LIN {X 0,Y 516.913,Z 376.098,A -85,B 0,C 180,E1 -4916.12,E2 -4916.12} C_VEL
LIN {X 0,Y 516.895,Z 376.101,A -85,B 0,C 180,E1 -4918.935,E2 -4918.935} C_VEL
LIN {X 0,Y 516.92,Z 376.096,A -85,B 0,C 180,E1 -4921.584,E2 -4921.584} C_VEL
LIN {X 0,Y 516.937,Z 376.095,A -85,B 0,C 180,E1 -4924.21,E2 -4924.21} C_VEL
LIN {X 0,Y 516.871,Z 376.104,A -85,B 0,C 180,E1 -4926.775,E2 -4926.775} C_VEL
LIN {X 0,Y 516.945,Z 376.094,A -85,B 0,C 180,E1 -4929.731,E2 -4929.731} C_VEL
LIN {X 0,Y 516.925,Z 376.098,A -85,B 0,C 180,E1 -4932.595,E2 -4932.595} C_VEL
LIN {X 0,Y 516.947,Z 376.094,A -85,B 0,C 180,E1 -4935.029,E2 -4935.029} C_VEL
LIN {X 0,Y 516.884,Z 376.104,A -85,B 0,C 180,E1 -4938.231,E2 -4938.231} C_VEL
LIN {X 0,Y 516.594,Z 376.439,A -85,B 0,C 180,E1 -4940.603,E2 -4940.603} C_VEL
LIN {X 0,Y 516.577,Z 379.88,A -85,B 0,C 180,E1 -4943.75,E2 -4943.75} C_VEL
LIN {X 0,Y 516.567,Z 382.466,A -85,B 0,C 180,E1 -4946.098,E2 -4946.098} C_VEL
LIN {X 0,Y 516.432,Z 386.765,A -85,B 0,C 180,E1 -4949.999,E2 -4949.999} C_VEL
LIN {X 0,Y 516.446,Z 391.091,A -85,B 0,C 180,E1 -4953.9,E2 -4953.9} C_VEL
LIN {X 0,Y 516.401,Z 394.057,A -85,B 0,C 180,E1 -4956.536,E2 -4956.536} C_VEL
LIN {X 0,Y 516.278,Z 397.014,A -85,B 0,C 180,E1 -4959.202,E2 -4959.202} C_VEL
LIN {X 0,Y 518.475,Z 408.871,A -85,B 0,C 180,E1 -4959.581,E2 -4959.581} C_VEL
LIN {X 0,Y 518.24,Z 422.351,A -85,B 0,C 180,E1 -4960.103,E2 -4960.103} C_VEL
LIN {X 0,Y 517.891,Z 434.499,A -85,B 0,C 180,E1 -4960.752,E2 -4960.752} C_VEL
LIN {X 0,Y 517.599,Z 446.016,A -85,B 0,C 180,E1 -4961.551,E2 -4961.551} C_VEL
LIN {X 0,Y 517.28,Z 455.69,A -85,B 0,C 180,E1 -4962.386,E2 -4962.386} C_VEL
LIN {X 0,Y 517.014,Z 464.898,A -85,B 0,C 180,E1 -4963.359,E2 -4963.359} C_VEL
LIN {X 0,Y 516.749,Z 474.087,A -85,B 0,C 180,E1 -4964.571,E2 -4964.571} C_VEL
LIN {X 0,Y 516.599,Z 481.479,A -85,B 0,C 180,E1 -4965.787,E2 -4965.787} C_VEL
LIN {X 0,Y 516.454,Z 487.37,A -85,B 0,C 180,E1 -4967.01,E2 -4967.01} C_VEL
LIN {X 0,Y 516.35,Z 491.98,A -85,B 0,C 180,E1 -4968.241,E2 -4968.241} C_VEL
LIN {X 0,Y 516.29,Z 494.408,A -85,B 0,C 180,E1 -4969.067,E2 -4969.067} C_VEL
LIN {X 0,Y 516.231,Z 496.687,A -85,B 0,C 180,E1 -4970.054,E2 -4970.054} C_VEL
LIN {X 0,Y 516.201,Z 498.869,A -85,B 0,C 180,E1 -4971.566,E2 -4971.566} C_VEL
LIN {X 0,Y 516.214,Z 499.464,A -85,B 0,C 180,E1 -4972.406,E2 -4972.406} C_VEL
LIN {X 0,Y 516.183,Z 499.561,A -85,B 0,C 180,E1 -4973.254,E2 -4973.254} C_VEL
LIN {X 0,Y 516.199,Z 499.165,A -85,B 0,C 180,E1 -4974.189,E2 -4974.189} C_VEL
LIN {X 0,Y 516.2,Z 498.417,A -85,B 0,C 180,E1 -4974.963,E2 -4974.963} C_VEL
LIN {X 0,Y 516.222,Z 496.702,A -85,B 0,C 180,E1 -4976.033,E2 -4976.033} C_VEL
LIN {X 0,Y 516.305,Z 494.141,A -85,B 0,C 180,E1 -4977.127,E2 -4977.127} C_VEL
LIN {X 0,Y 516.383,Z 489.92,A -85,B 0,C 180,E1 -4978.445,E2 -4978.445} C_VEL
LIN {X 0,Y 516.516,Z 484.125,A -85,B 0,C 180,E1 -4979.794,E2 -4979.794} C_VEL
LIN {X 0,Y 516.715,Z 476.736,A -85,B 0,C 180,E1 -4981.119,E2 -4981.119} C_VEL
LIN {X 0,Y 516.92,Z 469.222,A -85,B 0,C 180,E1 -4982.2,E2 -4982.2} C_VEL
LIN {X 0,Y 517.194,Z 460.061,A -85,B 0,C 180,E1 -4983.271,E2 -4983.271} C_VEL
LIN {X 0,Y 517.481,Z 449.897,A -85,B 0,C 180,E1 -4984.228,E2 -4984.228} C_VEL
LIN {X 0,Y 517.778,Z 439.926,A -85,B 0,C 180,E1 -4984.989,E2 -4984.989} C_VEL
LIN {X 0,Y 518.075,Z 428.588,A -85,B 0,C 180,E1 -4985.682,E2 -4985.682} C_VEL
LIN {X 0,Y 518.328,Z 415.979,A -85,B 0,C 180,E1 -4986.262,E2 -4986.262} C_VEL
LIN {X 0,Y 518.286,Z 407.164,A -85,B 0,C 180,E1 -4986.574,E2 -4986.574} C_VEL
LIN {X 0,Y 516.296,Z 397.126,A -85,B 0,C 180,E1 -4986.895,E2 -4986.895} C_VEL
LIN {X 0,Y 516.309,Z 393.355,A -85,B 0,C 180,E1 -4990.335,E2 -4990.335} C_VEL
LIN {X 0,Y 516.37,Z 390.564,A -85,B 0,C 180,E1 -4992.881,E2 -4992.881} C_VEL
LIN {X 0,Y 516.411,Z 388.218,A -85,B 0,C 180,E1 -4995.044,E2 -4995.044} C_VEL
LIN {X 0,Y 516.446,Z 384.839,A -85,B 0,C 180,E1 -4998.179,E2 -4998.179} C_VEL
LIN {X 0,Y 516.457,Z 381.512,A -85,B 0,C 180,E1 -5001.246,E2 -5001.246} C_VEL
LIN {X 0,Y 516.553,Z 378.293,A -85,B 0,C 180,E1 -5004.194,E2 -5004.194} C_VEL
LIN {X 0,Y 516.601,Z 376.21,A -85,B 0,C 180,E1 -5006.098,E2 -5006.098} C_VEL
LIN {X 0,Y 516.861,Z 376.104,A -85,B 0,C 180,E1 -5008.937,E2 -5008.937} C_VEL
LIN {X 0,Y 516.907,Z 376.097,A -85,B 0,C 180,E1 -5011.584,E2 -5011.584} C_VEL
LIN {X 0,Y 516.915,Z 376.097,A -85,B 0,C 180,E1 -5014.21,E2 -5014.21} C_VEL
LIN {X 0,Y 516.885,Z 376.101,A -85,B 0,C 180,E1 -5016.777,E2 -5016.777} C_VEL
LIN {X 0,Y 516.92,Z 376.095,A -85,B 0,C 180,E1 -5019.73,E2 -5019.73} C_VEL
LIN {X 0,Y 516.911,Z 376.096,A -85,B 0,C 180,E1 -5022.596,E2 -5022.596} C_VEL
LIN {X 0,Y 516.921,Z 376.095,A -85,B 0,C 180,E1 -5025.03,E2 -5025.03} C_VEL
LIN {X 0,Y 516.983,Z 376.088,A -85,B 0,C 180,E1 -5028.234,E2 -5028.234} C_VEL
LIN {X 0,Y 516.953,Z 376.094,A -85,B 0,C 180,E1 -5031.399,E2 -5031.399} C_VEL
LIN {X 0,Y 517.047,Z 376.08,A -85,B 0,C 180,E1 -5034.54,E2 -5034.54} C_VEL
LIN {X 0,Y 517.07,Z 376.077,A -85,B 0,C 180,E1 -5037.663,E2 -5037.663} C_VEL
LIN {X 0,Y 517.077,Z 376.079,A -85,B 0,C 180,E1 -5040.779,E2 -5040.779} C_VEL
LIN {X 0,Y 517.026,Z 376.083,A -85,B 0,C 180,E1 -5043.117,E2 -5043.117} C_VEL
LIN {X 0,Y 516.991,Z 376.09,A -85,B 0,C 180,E1 -5046.243,E2 -5046.243} C_VEL
LIN {X 0,Y 516.937,Z 376.093,A -85,B 0,C 180,E1 -5049.39,E2 -5049.39} C_VEL
LIN {X 0,Y 516.962,Z 376.092,A -85,B 0,C 180,E1 -5051.825,E2 -5051.825} C_VEL
LIN {X 0,Y 516.923,Z 376.095,A -85,B 0,C 180,E1 -5055.147,E2 -5055.147} C_VEL
LIN {X 0,Y 516.907,Z 376.1,A -85,B 0,C 180,E1 -5058.223,E2 -5058.223} C_VEL
LIN {X 0,Y 516.898,Z 376.099,A -85,B 0,C 180,E1 -5060.702,E2 -5060.702} C_VEL
LIN {X 0,Y 516.888,Z 376.1,A -85,B 0,C 180,E1 -5063.223,E2 -5063.223} C_VEL
LIN {X 0,Y 516.926,Z 376.098,A -85,B 0,C 180,E1 -5066.198,E2 -5066.198} C_VEL
LIN {X 0,Y 516.905,Z 376.101,A -85,B 0,C 180,E1 -5069.306,E2 -5069.306} C_VEL
LIN {X 0,Y 516.884,Z 376.1,A -85,B 0,C 180,E1 -5072.546,E2 -5072.546} C_VEL
LIN {X 0,Y 516.868,Z 376.102,A -85,B 0,C 180,E1 -5075.334,E2 -5075.334} C_VEL
LIN {X 0,Y 516.869,Z 376.102,A -85,B 0,C 180,E1 -5077.945,E2 -5077.945} C_VEL
LIN {X 0,Y 516.894,Z 376.101,A -85,B 0,C 180,E1 -5080.741,E2 -5080.741} C_VEL
LIN {X 0,Y 516.869,Z 376.108,A -85,B 0,C 180,E1 -5083.905,E2 -5083.905} C_VEL
LIN {X 0,Y 516.87,Z 376.106,A -85,B 0,C 180,E1 -5086.109,E2 -5086.109} C_VEL
LIN {X 0,Y 516.894,Z 376.103,A -85,B 0,C 180,E1 -5089.262,E2 -5089.262} C_VEL
LIN {X 0,Y 516.908,Z 376.193,A -85,B 0,C 180,E1 -5091.229,E2 -5091.229} C_VEL
LIN {X 0,Y 518.065,Z 382.766,A -85,B 0,C 180,E1 -5093.838,E2 -5093.838} C_VEL
LIN {X 0,Y 518.075,Z 388.22,A -85,B 0,C 180,E1 -5095.843,E2 -5095.843} C_VEL
LIN {X 0,Y 517.76,Z 397.502,A -85,B 0,C 180,E1 -5098.951,E2 -5098.951} C_VEL
LIN {X 0,Y 517.58,Z 406.694,A -85,B 0,C 180,E1 -5101.959,E2 -5101.959} C_VEL
LIN {X 0,Y 517.315,Z 414.964,A -85,B 0,C 180,E1 -5104.665,E2 -5104.665} C_VEL
LIN {X 0,Y 517.11,Z 424.231,A -85,B 0,C 180,E1 -5107.635,E2 -5107.635} C_VEL
LIN {X 0,Y 516.902,Z 433.498,A -85,B 0,C 180,E1 -5110.544,E2 -5110.544} C_VEL
LIN {X 0,Y 516.709,Z 442.766,A -85,B 0,C 180,E1 -5113.405,E2 -5113.405} C_VEL
LIN {X 0,Y 516.577,Z 451.536,A -85,B 0,C 180,E1 -5116.078,E2 -5116.078} C_VEL
LIN {X 0,Y 518.522,Z 464.249,A -85,B 0,C 180,E1 -5116.431,E2 -5116.431} C_VEL
LIN {X 0,Y 518.314,Z 475.818,A -85,B 0,C 180,E1 -5116.824,E2 -5116.824} C_VEL
LIN {X 0,Y 517.995,Z 487.442,A -85,B 0,C 180,E1 -5117.364,E2 -5117.364} C_VEL
LIN {X 0,Y 517.684,Z 499.584,A -85,B 0,C 180,E1 -5118.11,E2 -5118.11} C_VEL
LIN {X 0,Y 517.42,Z 510.283,A -85,B 0,C 180,E1 -5118.941,E2 -5118.941} C_VEL
LIN {X 0,Y 517.081,Z 519.555,A -85,B 0,C 180,E1 -5119.825,E2 -5119.825} C_VEL
LIN {X 0,Y 516.866,Z 528.004,A -85,B 0,C 180,E1 -5120.808,E2 -5120.808} C_VEL
LIN {X 0,Y 516.639,Z 536.247,A -85,B 0,C 180,E1 -5121.987,E2 -5121.987} C_VEL
LIN {X 0,Y 516.478,Z 543.085,A -85,B 0,C 180,E1 -5123.203,E2 -5123.203} C_VEL
LIN {X 0,Y 516.405,Z 548.956,A -85,B 0,C 180,E1 -5124.535,E2 -5124.535} C_VEL
LIN {X 0,Y 516.343,Z 552.899,A -85,B 0,C 180,E1 -5125.708,E2 -5125.708} C_VEL
LIN {X 0,Y 516.282,Z 555.811,A -85,B 0,C 180,E1 -5126.88,E2 -5126.88} C_VEL
LIN {X 0,Y 516.261,Z 557.199,A -85,B 0,C 180,E1 -5127.661,E2 -5127.661} C_VEL
LIN {X 0,Y 516.16,Z 558.786,A -85,B 0,C 180,E1 -5129.221,E2 -5129.221} C_VEL
LIN {X 0,Y 516.154,Z 559,A -85,B 0,C 180,E1 -5130.001,E2 -5130.001} C_VEL
LIN {X 0,Y 516.192,Z 558.184,A -85,B 0,C 180,E1 -5131.562,E2 -5131.562} C_VEL
LIN {X 0,Y 516.262,Z 557.196,A -85,B 0,C 180,E1 -5132.342,E2 -5132.342} C_VEL
LIN {X 0,Y 516.283,Z 555.807,A -85,B 0,C 180,E1 -5133.123,E2 -5133.123} C_VEL
LIN {X 0,Y 516.344,Z 552.892,A -85,B 0,C 180,E1 -5134.295,E2 -5134.295} C_VEL
LIN {X 0,Y 516.406,Z 548.944,A -85,B 0,C 180,E1 -5135.468,E2 -5135.468} C_VEL
LIN {X 0,Y 516.488,Z 543.025,A -85,B 0,C 180,E1 -5136.809,E2 -5136.809} C_VEL
LIN {X 0,Y 516.642,Z 536.228,A -85,B 0,C 180,E1 -5138.016,E2 -5138.016} C_VEL
LIN {X 0,Y 516.871,Z 527.981,A -85,B 0,C 180,E1 -5139.195,E2 -5139.195} C_VEL
LIN {X 0,Y 517.08,Z 519.526,A -85,B 0,C 180,E1 -5140.178,E2 -5140.178} C_VEL
LIN {X 0,Y 517.434,Z 509.081,A -85,B 0,C 180,E1 -5141.161,E2 -5141.161} C_VEL
LIN {X 0,Y 517.7,Z 497.781,A -85,B 0,C 180,E1 -5142.016,E2 -5142.016} C_VEL
LIN {X 0,Y 517.992,Z 487.386,A -85,B 0,C 180,E1 -5142.639,E2 -5142.639} C_VEL
LIN {X 0,Y 518.284,Z 475.731,A -85,B 0,C 180,E1 -5143.179,E2 -5143.179} C_VEL
LIN {X 0,Y 518.421,Z 462.758,A -85,B 0,C 180,E1 -5143.613,E2 -5143.613} C_VEL
LIN {X 0,Y 516.577,Z 451.526,A -85,B 0,C 180,E1 -5143.925,E2 -5143.925} C_VEL
LIN {X 0,Y 516.715,Z 442.755,A -85,B 0,C 180,E1 -5146.598,E2 -5146.598} C_VEL
LIN {X 0,Y 516.91,Z 433.488,A -85,B 0,C 180,E1 -5149.459,E2 -5149.459} C_VEL
LIN {X 0,Y 517.102,Z 423.961,A -85,B 0,C 180,E1 -5152.452,E2 -5152.452} C_VEL
LIN {X 0,Y 517.376,Z 413.63,A -85,B 0,C 180,E1 -5155.766,E2 -5155.766} C_VEL
LIN {X 0,Y 517.604,Z 404.3,A -85,B 0,C 180,E1 -5158.818,E2 -5158.818} C_VEL
LIN {X 0,Y 517.882,Z 394.893,A -85,B 0,C 180,E1 -5161.956,E2 -5161.956} C_VEL
LIN {X 0,Y 518.147,Z 386.815,A -85,B 0,C 180,E1 -5164.729,E2 -5164.729} C_VEL
LIN {X 0,Y 518.059,Z 382.767,A -85,B 0,C 180,E1 -5166.167,E2 -5166.167} C_VEL
LIN {X 0,Y 516.886,Z 376.104,A -85,B 0,C 180,E1 -5168.836,E2 -5168.836} C_VEL
LIN {X 0,Y 516.917,Z 376.097,A -85,B 0,C 180,E1 -5171.776,E2 -5171.776} C_VEL
LIN {X 0,Y 516.901,Z 376.1,A -85,B 0,C 180,E1 -5175.007,E2 -5175.007} C_VEL
LIN {X 0,Y 516.919,Z 376.098,A -85,B 0,C 180,E1 -5178.399,E2 -5178.399} C_VEL
LIN {X 0,Y 516.885,Z 376.102,A -85,B 0,C 180,E1 -5181.284,E2 -5181.284} C_VEL
LIN {X 0,Y 516.876,Z 376.103,A -85,B 0,C 180,E1 -5184.22,E2 -5184.22} C_VEL
LIN {X 0,Y 516.886,Z 376.102,A -85,B 0,C 180,E1 -5187.052,E2 -5187.052} C_VEL
LIN {X 0,Y 516.897,Z 376.099,A -85,B 0,C 180,E1 -5189.796,E2 -5189.796} C_VEL
LIN {X 0,Y 516.93,Z 376.096,A -85,B 0,C 180,E1 -5192.467,E2 -5192.467} C_VEL
LIN {X 0,Y 516.913,Z 376.099,A -85,B 0,C 180,E1 -5195.072,E2 -5195.072} C_VEL
LIN {X 0,Y 516.89,Z 376.102,A -85,B 0,C 180,E1 -5198.462,E2 -5198.462} C_VEL
LIN {X 0,Y 516.907,Z 376.099,A -85,B 0,C 180,E1 -5200.955,E2 -5200.955} C_VEL
LIN {X 0,Y 516.918,Z 376.097,A -85,B 0,C 180,E1 -5203.41,E2 -5203.41} C_VEL
LIN {X 0,Y 516.899,Z 376.1,A -85,B 0,C 180,E1 -5205.834,E2 -5205.834} C_VEL
LIN {X 0,Y 516.97,Z 376.091,A -85,B 0,C 180,E1 -5208.234,E2 -5208.234} C_VEL
LIN {X 0,Y 516.974,Z 376.089,A -85,B 0,C 180,E1 -5211.4,E2 -5211.4} C_VEL
LIN {X 0,Y 517.013,Z 376.086,A -85,B 0,C 180,E1 -5213.757,E2 -5213.757} C_VEL
LIN {X 0,Y 517.087,Z 376.076,A -85,B 0,C 180,E1 -5217.663,E2 -5217.663} C_VEL
LIN {X 0,Y 517.095,Z 376.075,A -85,B 0,C 180,E1 -5220.779,E2 -5220.779} C_VEL
LIN {X 0,Y 517.016,Z 376.085,A -85,B 0,C 180,E1 -5223.117,E2 -5223.117} C_VEL
LIN {X 0,Y 517.007,Z 376.088,A -85,B 0,C 180,E1 -5226.243,E2 -5226.243} C_VEL
LIN {X 0,Y 516.957,Z 376.093,A -85,B 0,C 180,E1 -5229.389,E2 -5229.389} C_VEL
LIN {X 0,Y 516.956,Z 376.093,A -85,B 0,C 180,E1 -5231.807,E2 -5231.807} C_VEL
LIN {X 0,Y 516.949,Z 376.093,A -85,B 0,C 180,E1 -5235.146,E2 -5235.146} C_VEL
LIN {X 0,Y 516.928,Z 376.096,A -85,B 0,C 180,E1 -5238.222,E2 -5238.222} C_VEL
LIN {X 0,Y 516.916,Z 376.098,A -85,B 0,C 180,E1 -5240.701,E2 -5240.701} C_VEL
LIN {X 0,Y 516.908,Z 376.099,A -85,B 0,C 180,E1 -5244.072,E2 -5244.072} C_VEL
LIN {X 0,Y 516.93,Z 376.094,A -85,B 0,C 180,E1 -5246.658,E2 -5246.658} C_VEL
LIN {X 0,Y 516.915,Z 376.098,A -85,B 0,C 180,E1 -5249.523,E2 -5249.523} C_VEL
LIN {X 0,Y 516.9,Z 376.099,A -85,B 0,C 180,E1 -5252.543,E2 -5252.543} C_VEL
LIN {X 0,Y 516.87,Z 376.106,A -85,B 0,C 180,E1 -5255.329,E2 -5255.329} C_VEL
LIN {X 0,Y 516.884,Z 376.101,A -85,B 0,C 180,E1 -5257.942,E2 -5257.942} C_VEL
LIN {X 0,Y 516.887,Z 376.102,A -85,B 0,C 180,E1 -5260.741,E2 -5260.741} C_VEL
LIN {X 0,Y 516.887,Z 376.102,A -85,B 0,C 180,E1 -5262.831,E2 -5262.831} C_VEL
LIN {X 0,Y 516.9,Z 376.1,A -85,B 0,C 180,E1 -5265.007,E2 -5265.007} C_VEL
LIN {X 0,Y 516.92,Z 376.096,A -85,B 0,C 180,E1 -5268.398,E2 -5268.398} C_VEL
LIN {X 0,Y 516.887,Z 376.1,A -85,B 0,C 180,E1 -5270.301,E2 -5270.301} C_VEL
LIN {X 0,Y 516.216,Z 376.187,A -85,B 0,C 180,E1 -5270.951,E2 -5270.951} C_VEL
LIN {X 0,Y 513.369,Z 376.542,A -85,B 0,C 180,E1 -5272.007,E2 -5272.007} C_VEL
LIN {X 0,Y 510.959,Z 376.843,A -85,B 0,C 180,E1 -5272.857,E2 -5272.857} C_VEL
LIN {X 0,Y 509.915,Z 376.971,A -85,B 0,C 180,E1 -5273.514,E2 -5273.514} C_VEL
LIN {X 0,Y 509.825,Z 376.981,A -85,B 0,C 180,E1 -5273.736,E2 -5273.736} C_VEL
LIN {X 0,Y 509.864,Z 376.976,A -85,B 0,C 180,E1 -5276.538,E2 -5276.538} C_VEL
LIN {X 0,Y 509.848,Z 376.978,A -85,B 0,C 180,E1 -5279.333,E2 -5279.333} C_VEL
LIN {X 0,Y 509.895,Z 376.971,A -85,B 0,C 180,E1 -5282.054,E2 -5282.054} C_VEL
LIN {X 0,Y 509.882,Z 376.974,A -85,B 0,C 180,E1 -5284.703,E2 -5284.703} C_VEL
LIN {X 0,Y 509.832,Z 376.98,A -85,B 0,C 180,E1 -5287.457,E2 -5287.457} C_VEL
LIN {X 0,Y 509.922,Z 376.968,A -85,B 0,C 180,E1 -5289.844,E2 -5289.844} C_VEL
LIN {X 0,Y 509.885,Z 376.973,A -85,B 0,C 180,E1 -5293.174,E2 -5293.174} C_VEL
LIN {X 0,Y 509.867,Z 376.975,A -85,B 0,C 180,E1 -5295.633,E2 -5295.633} C_VEL
LIN {X 0,Y 509.848,Z 376.98,A -85,B 0,C 180,E1 -5298.154,E2 -5298.154} C_VEL
LIN {X 0,Y 509.521,Z 377.021,A -85,B 0,C 180,E1 -5300.471,E2 -5300.471} C_VEL
LIN {X 0,Y 509.527,Z 380.47,A -85,B 0,C 180,E1 -5303.663,E2 -5303.663} C_VEL
LIN {X 0,Y 509.519,Z 383.053,A -85,B 0,C 180,E1 -5306.044,E2 -5306.044} C_VEL
LIN {X 0,Y 509.359,Z 387.412,A -85,B 0,C 180,E1 -5309.998,E2 -5309.998} C_VEL
LIN {X 0,Y 509.371,Z 391.778,A -85,B 0,C 180,E1 -5313.954,E2 -5313.954} C_VEL
LIN {X 0,Y 509.347,Z 394.758,A -85,B 0,C 180,E1 -5316.555,E2 -5316.555} C_VEL
LIN {X 0,Y 509.21,Z 397.44,A -85,B 0,C 180,E1 -5319.006,E2 -5319.006} C_VEL
LIN {X 0,Y 511.522,Z 409.074,A -85,B 0,C 180,E1 -5319.388,E2 -5319.388} C_VEL
LIN {X 0,Y 511.364,Z 421.956,A -85,B 0,C 180,E1 -5319.89,E2 -5319.89} C_VEL
LIN {X 0,Y 511.001,Z 433.55,A -85,B 0,C 180,E1 -5320.498,E2 -5320.498} C_VEL
LIN {X 0,Y 510.697,Z 445.317,A -85,B 0,C 180,E1 -5321.307,E2 -5321.307} C_VEL
LIN {X 0,Y 510.32,Z 455.958,A -85,B 0,C 180,E1 -5322.225,E2 -5322.225} C_VEL
LIN {X 0,Y 510.067,Z 464.568,A -85,B 0,C 180,E1 -5323.139,E2 -5323.139} C_VEL
LIN {X 0,Y 509.792,Z 472.538,A -85,B 0,C 180,E1 -5324.162,E2 -5324.162} C_VEL
LIN {X 0,Y 509.595,Z 480.277,A -85,B 0,C 180,E1 -5325.394,E2 -5325.394} C_VEL
LIN {X 0,Y 509.425,Z 485.575,A -85,B 0,C 180,E1 -5326.426,E2 -5326.426} C_VEL
LIN {X 0,Y 509.304,Z 491.125,A -85,B 0,C 180,E1 -5327.797,E2 -5327.797} C_VEL
LIN {X 0,Y 509.224,Z 494.601,A -85,B 0,C 180,E1 -5328.923,E2 -5328.923} C_VEL
LIN {X 0,Y 509.134,Z 497.43,A -85,B 0,C 180,E1 -5330.186,E2 -5330.186} C_VEL
LIN {X 0,Y 509.119,Z 498.746,A -85,B 0,C 180,E1 -5331.031,E2 -5331.031} C_VEL
LIN {X 0,Y 509.123,Z 499.873,A -85,B 0,C 180,E1 -5332.35,E2 -5332.35} C_VEL
LIN {X 0,Y 509.104,Z 499.927,A -85,B 0,C 180,E1 -5333.597,E2 -5333.597} C_VEL
LIN {X 0,Y 509.106,Z 499.39,A -85,B 0,C 180,E1 -5334.463,E2 -5334.463} C_VEL
LIN {X 0,Y 509.107,Z 498.37,A -85,B 0,C 180,E1 -5335.335,E2 -5335.335} C_VEL
LIN {X 0,Y 509.192,Z 495.915,A -85,B 0,C 180,E1 -5336.65,E2 -5336.65} C_VEL
LIN {X 0,Y 509.275,Z 492.238,A -85,B 0,C 180,E1 -5337.98,E2 -5337.98} C_VEL
LIN {X 0,Y 509.401,Z 487.436,A -85,B 0,C 180,E1 -5339.259,E2 -5339.259} C_VEL
LIN {X 0,Y 509.569,Z 480.412,A -85,B 0,C 180,E1 -5340.682,E2 -5340.682} C_VEL
LIN {X 0,Y 509.823,Z 473.326,A -85,B 0,C 180,E1 -5341.82,E2 -5341.82} C_VEL
LIN {X 0,Y 510.065,Z 465.228,A -85,B 0,C 180,E1 -5342.883,E2 -5342.883} C_VEL
LIN {X 0,Y 510.398,Z 455.733,A -85,B 0,C 180,E1 -5343.892,E2 -5343.892} C_VEL
LIN {X 0,Y 510.72,Z 444.893,A -85,B 0,C 180,E1 -5344.823,E2 -5344.823} C_VEL
LIN {X 0,Y 511.012,Z 434.442,A -85,B 0,C 180,E1 -5345.542,E2 -5345.542} C_VEL
LIN {X 0,Y 511.318,Z 423.016,A -85,B 0,C 180,E1 -5346.159,E2 -5346.159} C_VEL
LIN {X 0,Y 511.585,Z 410.272,A -85,B 0,C 180,E1 -5346.664,E2 -5346.664} C_VEL
LIN {X 0,Y 510.149,Z 401.591,A -85,B 0,C 180,E1 -5346.962,E2 -5346.962} C_VEL
LIN {X 0,Y 509.214,Z 397.595,A -85,B 0,C 180,E1 -5347.084,E2 -5347.084} C_VEL
LIN {X 0,Y 509.252,Z 393.912,A -85,B 0,C 180,E1 -5350.435,E2 -5350.435} C_VEL
LIN {X 0,Y 509.339,Z 390.438,A -85,B 0,C 180,E1 -5353.62,E2 -5353.62} C_VEL
LIN {X 0,Y 509.364,Z 387.478,A -85,B 0,C 180,E1 -5356.379,E2 -5356.379} C_VEL
LIN {X 0,Y 509.401,Z 384.264,A -85,B 0,C 180,E1 -5359.356,E2 -5359.356} C_VEL
LIN {X 0,Y 509.453,Z 380.728,A -85,B 0,C 180,E1 -5362.628,E2 -5362.628} C_VEL
LIN {X 0,Y 509.527,Z 377.543,A -85,B 0,C 180,E1 -5365.562,E2 -5365.562} C_VEL
LIN {X 0,Y 509.574,Z 377.015,A -85,B 0,C 180,E1 -5366.518,E2 -5366.518} C_VEL
LIN {X 0,Y 509.823,Z 376.982,A -85,B 0,C 180,E1 -5369.333,E2 -5369.333} C_VEL
LIN {X 0,Y 509.877,Z 376.974,A -85,B 0,C 180,E1 -5372.054,E2 -5372.054} C_VEL
LIN {X 0,Y 509.865,Z 376.976,A -85,B 0,C 180,E1 -5374.703,E2 -5374.703} C_VEL
LIN {X 0,Y 509.864,Z 376.976,A -85,B 0,C 180,E1 -5377.441,E2 -5377.441} C_VEL
LIN {X 0,Y 509.897,Z 376.969,A -85,B 0,C 180,E1 -5379.844,E2 -5379.844} C_VEL
LIN {X 0,Y 509.867,Z 376.978,A -85,B 0,C 180,E1 -5383.174,E2 -5383.174} C_VEL
LIN {X 0,Y 509.845,Z 376.978,A -85,B 0,C 180,E1 -5385.634,E2 -5385.634} C_VEL
LIN {X 0,Y 509.907,Z 376.97,A -85,B 0,C 180,E1 -5388.874,E2 -5388.874} C_VEL
LIN {X 0,Y 509.931,Z 376.966,A -85,B 0,C 180,E1 -5392.078,E2 -5392.078} C_VEL
LIN {X 0,Y 509.993,Z 376.959,A -85,B 0,C 180,E1 -5394.464,E2 -5394.464} C_VEL
LIN {X 0,Y 510.04,Z 376.953,A -85,B 0,C 180,E1 -5397.631,E2 -5397.631} C_VEL
LIN {X 0,Y 510.047,Z 376.955,A -85,B 0,C 180,E1 -5400.79,E2 -5400.79} C_VEL
LIN {X 0,Y 509.967,Z 376.963,A -85,B 0,C 180,E1 -5403.16,E2 -5403.16} C_VEL
LIN {X 0,Y 509.959,Z 376.965,A -85,B 0,C 180,E1 -5406.33,E2 -5406.33} C_VEL
LIN {X 0,Y 509.897,Z 376.973,A -85,B 0,C 180,E1 -5408.721,E2 -5408.721} C_VEL
LIN {X 0,Y 509.93,Z 376.967,A -85,B 0,C 180,E1 -5411.931,E2 -5411.931} C_VEL
LIN {X 0,Y 509.873,Z 376.974,A -85,B 0,C 180,E1 -5415.243,E2 -5415.243} C_VEL
LIN {X 0,Y 509.869,Z 376.975,A -85,B 0,C 180,E1 -5418.002,E2 -5418.002} C_VEL
LIN {X 0,Y 509.843,Z 376.981,A -85,B 0,C 180,E1 -5421.002,E2 -5421.002} C_VEL
LIN {X 0,Y 509.848,Z 376.98,A -85,B 0,C 180,E1 -5423.563,E2 -5423.563} C_VEL
LIN {X 0,Y 509.895,Z 376.975,A -85,B 0,C 180,E1 -5426.38,E2 -5426.38} C_VEL
LIN {X 0,Y 509.86,Z 376.978,A -85,B 0,C 180,E1 -5428.845,E2 -5428.845} C_VEL
LIN {X 0,Y 509.809,Z 376.984,A -85,B 0,C 180,E1 -5431.591,E2 -5431.591} C_VEL
LIN {X 0,Y 509.838,Z 376.981,A -85,B 0,C 180,E1 -5434.415,E2 -5434.415} C_VEL
LIN {X 0,Y 509.807,Z 376.985,A -85,B 0,C 180,E1 -5437.342,E2 -5437.342} C_VEL
LIN {X 0,Y 509.849,Z 376.979,A -85,B 0,C 180,E1 -5440.381,E2 -5440.381} C_VEL
LIN {X 0,Y 509.826,Z 376.984,A -85,B 0,C 180,E1 -5443.066,E2 -5443.066} C_VEL
LIN {X 0,Y 509.818,Z 376.985,A -85,B 0,C 180,E1 -5445.794,E2 -5445.794} C_VEL
LIN {X 0,Y 509.856,Z 376.979,A -85,B 0,C 180,E1 -5448.578,E2 -5448.578} C_VEL
LIN {X 0,Y 509.898,Z 377.088,A -85,B 0,C 180,E1 -5450.974,E2 -5450.974} C_VEL
LIN {X 0,Y 511.094,Z 384.034,A -85,B 0,C 180,E1 -5453.754,E2 -5453.754} C_VEL
LIN {X 0,Y 511.056,Z 390.423,A -85,B 0,C 180,E1 -5456.157,E2 -5456.157} C_VEL
LIN {X 0,Y 510.757,Z 398.719,A -85,B 0,C 180,E1 -5458.971,E2 -5458.971} C_VEL
LIN {X 0,Y 510.521,Z 408.152,A -85,B 0,C 180,E1 -5462.094,E2 -5462.094} C_VEL
LIN {X 0,Y 510.294,Z 416.288,A -85,B 0,C 180,E1 -5464.728,E2 -5464.728} C_VEL
LIN {X 0,Y 510.074,Z 425.679,A -85,B 0,C 180,E1 -5467.776,E2 -5467.776} C_VEL
LIN {X 0,Y 509.855,Z 434.822,A -85,B 0,C 180,E1 -5470.683,E2 -5470.683} C_VEL
LIN {X 0,Y 509.645,Z 445.413,A -85,B 0,C 180,E1 -5473.992,E2 -5473.992} C_VEL
LIN {X 0,Y 509.523,Z 451.652,A -85,B 0,C 180,E1 -5475.897,E2 -5475.897} C_VEL
LIN {X 0,Y 511.593,Z 464.249,A -85,B 0,C 180,E1 -5476.243,E2 -5476.243} C_VEL
LIN {X 0,Y 511.38,Z 477.024,A -85,B 0,C 180,E1 -5476.693,E2 -5476.693} C_VEL
LIN {X 0,Y 511.019,Z 489.206,A -85,B 0,C 180,E1 -5477.29,E2 -5477.29} C_VEL
LIN {X 0,Y 510.724,Z 499.976,A -85,B 0,C 180,E1 -5477.973,E2 -5477.973} C_VEL
LIN {X 0,Y 510.395,Z 511.419,A -85,B 0,C 180,E1 -5478.887,E2 -5478.887} C_VEL
LIN {X 0,Y 510.028,Z 521.35,A -85,B 0,C 180,E1 -5479.883,E2 -5479.883} C_VEL
LIN {X 0,Y 509.759,Z 530.973,A -85,B 0,C 180,E1 -5481.079,E2 -5481.079} C_VEL
LIN {X 0,Y 509.52,Z 538.631,A -85,B 0,C 180,E1 -5482.273,E2 -5482.273} C_VEL
LIN {X 0,Y 509.335,Z 545.687,A -85,B 0,C 180,E1 -5483.664,E2 -5483.664} C_VEL
LIN {X 0,Y 509.247,Z 550.378,A -85,B 0,C 180,E1 -5484.855,E2 -5484.855} C_VEL
LIN {X 0,Y 509.253,Z 553.962,A -85,B 0,C 180,E1 -5486.045,E2 -5486.045} C_VEL
LIN {X 0,Y 509.2,Z 555.811,A -85,B 0,C 180,E1 -5486.837,E2 -5486.837} C_VEL
LIN {X 0,Y 509.161,Z 557.198,A -85,B 0,C 180,E1 -5487.628,E2 -5487.628} C_VEL
LIN {X 0,Y 509.073,Z 558.786,A -85,B 0,C 180,E1 -5489.211,E2 -5489.211} C_VEL
LIN {X 0,Y 509.065,Z 559,A -85,B 0,C 180,E1 -5490.002,E2 -5490.002} C_VEL
LIN {X 0,Y 509.113,Z 558.184,A -85,B 0,C 180,E1 -5491.584,E2 -5491.584} C_VEL
LIN {X 0,Y 509.162,Z 557.196,A -85,B 0,C 180,E1 -5492.375,E2 -5492.375} C_VEL
LIN {X 0,Y 509.201,Z 555.807,A -85,B 0,C 180,E1 -5493.166,E2 -5493.166} C_VEL
LIN {X 0,Y 509.234,Z 552.892,A -85,B 0,C 180,E1 -5494.355,E2 -5494.355} C_VEL
LIN {X 0,Y 509.345,Z 548.943,A -85,B 0,C 180,E1 -5495.544,E2 -5495.544} C_VEL
LIN {X 0,Y 509.412,Z 543.275,A -85,B 0,C 180,E1 -5496.855,E2 -5496.855} C_VEL
LIN {X 0,Y 509.586,Z 536.228,A -85,B 0,C 180,E1 -5498.128,E2 -5498.128} C_VEL
LIN {X 0,Y 509.847,Z 527.981,A -85,B 0,C 180,E1 -5499.322,E2 -5499.322} C_VEL
LIN {X 0,Y 510.071,Z 519.527,A -85,B 0,C 180,E1 -5500.32,E2 -5500.32} C_VEL
LIN {X 0,Y 510.464,Z 509.08,A -85,B 0,C 180,E1 -5501.316,E2 -5501.316} C_VEL
LIN {X 0,Y 510.733,Z 498.511,A -85,B 0,C 180,E1 -5502.131,E2 -5502.131} C_VEL
LIN {X 0,Y 511.051,Z 487.385,A -85,B 0,C 180,E1 -5502.813,E2 -5502.813} C_VEL
LIN {X 0,Y 511.364,Z 475.731,A -85,B 0,C 180,E1 -5503.361,E2 -5503.361} C_VEL
LIN {X 0,Y 511.436,Z 463.215,A -85,B 0,C 180,E1 -5503.789,E2 -5503.789} C_VEL
LIN {X 0,Y 509.536,Z 451.526,A -85,B 0,C 180,E1 -5504.122,E2 -5504.122} C_VEL
LIN {X 0,Y 509.721,Z 441.432,A -85,B 0,C 180,E1 -5507.245,E2 -5507.245} C_VEL
LIN {X 0,Y 509.927,Z 432.164,A -85,B 0,C 180,E1 -5510.156,E2 -5510.156} C_VEL
LIN {X 0,Y 510.114,Z 422.897,A -85,B 0,C 180,E1 -5513.121,E2 -5513.121} C_VEL
LIN {X 0,Y 510.373,Z 413.575,A -85,B 0,C 180,E1 -5516.146,E2 -5516.146} C_VEL
LIN {X 0,Y 510.619,Z 404.22,A -85,B 0,C 180,E1 -5519.25,E2 -5519.25} C_VEL
LIN {X 0,Y 510.92,Z 396.157,A -85,B 0,C 180,E1 -5521.979,E2 -5521.979} C_VEL
LIN {X 0,Y 511.186,Z 388.062,A -85,B 0,C 180,E1 -5524.796,E2 -5524.796} C_VEL
LIN {X 0,Y 511.081,Z 384.031,A -85,B 0,C 180,E1 -5526.251,E2 -5526.251} C_VEL
LIN {X 0,Y 509.866,Z 376.978,A -85,B 0,C 180,E1 -5529.16,E2 -5529.16} C_VEL
LIN {X 0,Y 509.861,Z 376.976,A -85,B 0,C 180,E1 -5531.897,E2 -5531.897} C_VEL
LIN {X 0,Y 509.845,Z 376.98,A -85,B 0,C 180,E1 -5534.67,E2 -5534.67} C_VEL
LIN {X 0,Y 509.838,Z 376.981,A -85,B 0,C 180,E1 -5537.51,E2 -5537.51} C_VEL
LIN {X 0,Y 509.85,Z 376.979,A -85,B 0,C 180,E1 -5540.648,E2 -5540.648} C_VEL
LIN {X 0,Y 509.83,Z 376.98,A -85,B 0,C 180,E1 -5543.647,E2 -5543.647} C_VEL
LIN {X 0,Y 509.846,Z 376.978,A -85,B 0,C 180,E1 -5546.538,E2 -5546.538} C_VEL
LIN {X 0,Y 509.85,Z 376.977,A -85,B 0,C 180,E1 -5549.334,E2 -5549.334} C_VEL
LIN {X 0,Y 509.896,Z 376.972,A -85,B 0,C 180,E1 -5552.055,E2 -5552.055} C_VEL
LIN {X 0,Y 509.881,Z 376.974,A -85,B 0,C 180,E1 -5554.704,E2 -5554.704} C_VEL
LIN {X 0,Y 509.831,Z 376.98,A -85,B 0,C 180,E1 -5557.458,E2 -5557.458} C_VEL
LIN {X 0,Y 509.922,Z 376.968,A -85,B 0,C 180,E1 -5559.845,E2 -5559.845} C_VEL
LIN {X 0,Y 509.889,Z 376.973,A -85,B 0,C 180,E1 -5563.175,E2 -5563.175} C_VEL
LIN {X 0,Y 509.868,Z 376.976,A -85,B 0,C 180,E1 -5565.634,E2 -5565.634} C_VEL
LIN {X 0,Y 509.917,Z 376.969,A -85,B 0,C 180,E1 -5568.875,E2 -5568.875} C_VEL
LIN {X 0,Y 509.956,Z 376.965,A -85,B 0,C 180,E1 -5572.078,E2 -5572.078} C_VEL
LIN {X 0,Y 509.984,Z 376.961,A -85,B 0,C 180,E1 -5574.464,E2 -5574.464} C_VEL
LIN {X 0,Y 510.058,Z 376.951,A -85,B 0,C 180,E1 -5577.631,E2 -5577.631} C_VEL
LIN {X 0,Y 510.066,Z 376.951,A -85,B 0,C 180,E1 -5580.789,E2 -5580.789} C_VEL
LIN {X 0,Y 509.958,Z 376.964,A -85,B 0,C 180,E1 -5583.16,E2 -5583.16} C_VEL
LIN {X 0,Y 509.958,Z 376.965,A -85,B 0,C 180,E1 -5586.33,E2 -5586.33} C_VEL
LIN {X 0,Y 509.92,Z 376.967,A -85,B 0,C 180,E1 -5588.72,E2 -5588.72} C_VEL
LIN {X 0,Y 509.909,Z 376.971,A -85,B 0,C 180,E1 -5591.932,E2 -5591.932} C_VEL
LIN {X 0,Y 509.899,Z 376.971,A -85,B 0,C 180,E1 -5595.242,E2 -5595.242} C_VEL
LIN {X 0,Y 509.886,Z 376.974,A -85,B 0,C 180,E1 -5597.998,E2 -5597.998} C_VEL
LIN {X 0,Y 509.854,Z 376.978,A -85,B 0,C 180,E1 -5601.002,E2 -5601.002} C_VEL
LIN {X 0,Y 509.869,Z 376.974,A -85,B 0,C 180,E1 -5604.426,E2 -5604.426} C_VEL
LIN {X 0,Y 509.889,Z 376.974,A -85,B 0,C 180,E1 -5607.055,E2 -5607.055} C_VEL
LIN {X 0,Y 509.862,Z 376.977,A -85,B 0,C 180,E1 -5609.751,E2 -5609.751} C_VEL
LIN {X 0,Y 509.877,Z 376.974,A -85,B 0,C 180,E1 -5612.774,E2 -5612.774} C_VEL
LIN {X 0,Y 509.83,Z 376.981,A -85,B 0,C 180,E1 -5615.578,E2 -5615.578} C_VEL
LIN {X 0,Y 509.854,Z 376.977,A -85,B 0,C 180,E1 -5618.338,E2 -5618.338} C_VEL
LIN {X 0,Y 509.86,Z 376.978,A -85,B 0,C 180,E1 -5621.425,E2 -5621.425} C_VEL
LIN {X 0,Y 509.844,Z 376.979,A -85,B 0,C 180,E1 -5624.669,E2 -5624.669} C_VEL
LIN {X 0,Y 509.862,Z 376.975,A -85,B 0,C 180,E1 -5628.103,E2 -5628.103} C_VEL
LIN {X 0,Y 509.852,Z 376.977,A -85,B 0,C 180,E1 -5630.647,E2 -5630.647} C_VEL
LIN {X 0,Y 509.825,Z 376.981,A -85,B 0,C 180,E1 -5633.736,E2 -5633.736} C_VEL
LIN {X 0,Y 509.158,Z 377.064,A -85,B 0,C 180,E1 -5634.396,E2 -5634.396} C_VEL
LIN {X 0,Y 506.346,Z 377.415,A -85,B 0,C 180,E1 -5635.468,E2 -5635.468} C_VEL
LIN {X 0,Y 503.959,Z 377.714,A -85,B 0,C 180,E1 -5636.331,E2 -5636.331} C_VEL
LIN {X 0,Y 502.911,Z 377.844,A -85,B 0,C 180,E1 -5636.998,E2 -5636.998} C_VEL
LIN {X 0,Y 502.813,Z 377.854,A -85,B 0,C 180,E1 -5637.223,E2 -5637.223} C_VEL
LIN {X 0,Y 502.819,Z 377.853,A -85,B 0,C 180,E1 -5640.064,E2 -5640.064} C_VEL
LIN {X 0,Y 502.836,Z 377.852,A -85,B 0,C 180,E1 -5642.532,E2 -5642.532} C_VEL
LIN {X 0,Y 502.832,Z 377.853,A -85,B 0,C 180,E1 -5645.298,E2 -5645.298} C_VEL
LIN {X 0,Y 502.786,Z 377.857,A -85,B 0,C 180,E1 -5647.826,E2 -5647.826} C_VEL
LIN {X 0,Y 502.83,Z 377.853,A -85,B 0,C 180,E1 -5650.399,E2 -5650.399} C_VEL
LIN {X 0,Y 502.833,Z 377.852,A -85,B 0,C 180,E1 -5652.93,E2 -5652.93} C_VEL
LIN {X 0,Y 502.849,Z 377.85,A -85,B 0,C 180,E1 -5655.428,E2 -5655.428} C_VEL
LIN {X 0,Y 502.817,Z 377.855,A -85,B 0,C 180,E1 -5658.072,E2 -5658.072} C_VEL
LIN {X 0,Y 502.491,Z 377.897,A -85,B 0,C 180,E1 -5660.337,E2 -5660.337} C_VEL
LIN {X 0,Y 502.456,Z 379.316,A -85,B 0,C 180,E1 -5661.958,E2 -5661.958} C_VEL
LIN {X 0,Y 502.413,Z 381.943,A -85,B 0,C 180,E1 -5664.379,E2 -5664.379} C_VEL
LIN {X 0,Y 502.472,Z 383.682,A -85,B 0,C 180,E1 -5665.988,E2 -5665.988} C_VEL
LIN {X 0,Y 502.287,Z 388.071,A -85,B 0,C 180,E1 -5669.998,E2 -5669.998} C_VEL
LIN {X 0,Y 502.299,Z 392.465,A -85,B 0,C 180,E1 -5674.01,E2 -5674.01} C_VEL
LIN {X 0,Y 502.274,Z 395.344,A -85,B 0,C 180,E1 -5676.557,E2 -5676.557} C_VEL
LIN {X 0,Y 502.169,Z 397.863,A -85,B 0,C 180,E1 -5678.803,E2 -5678.803} C_VEL
LIN {X 0,Y 504.504,Z 409.378,A -85,B 0,C 180,E1 -5679.192,E2 -5679.192} C_VEL
LIN {X 0,Y 504.542,Z 420.401,A -85,B 0,C 180,E1 -5679.621,E2 -5679.621} C_VEL
LIN {X 0,Y 504.121,Z 432.469,A -85,B 0,C 180,E1 -5680.237,E2 -5680.237} C_VEL
LIN {X 0,Y 503.816,Z 443.296,A -85,B 0,C 180,E1 -5680.955,E2 -5680.955} C_VEL
LIN {X 0,Y 503.505,Z 453.241,A -85,B 0,C 180,E1 -5681.777,E2 -5681.777} C_VEL
LIN {X 0,Y 503.189,Z 462.224,A -85,B 0,C 180,E1 -5682.685,E2 -5682.685} C_VEL
LIN {X 0,Y 502.853,Z 470.814,A -85,B 0,C 180,E1 -5683.743,E2 -5683.743} C_VEL
LIN {X 0,Y 502.618,Z 478.471,A -85,B 0,C 180,E1 -5684.899,E2 -5684.899} C_VEL
LIN {X 0,Y 502.44,Z 484.588,A -85,B 0,C 180,E1 -5686.035,E2 -5686.035} C_VEL
LIN {X 0,Y 502.313,Z 489.184,A -85,B 0,C 180,E1 -5687.085,E2 -5687.085} C_VEL
LIN {X 0,Y 502.218,Z 493.576,A -85,B 0,C 180,E1 -5688.351,E2 -5688.351} C_VEL
LIN {X 0,Y 502.096,Z 496.848,A -85,B 0,C 180,E1 -5689.627,E2 -5689.627} C_VEL
LIN {X 0,Y 502.038,Z 498.455,A -85,B 0,C 180,E1 -5690.484,E2 -5690.484} C_VEL
LIN {X 0,Y 502.053,Z 499.549,A -85,B 0,C 180,E1 -5691.342,E2 -5691.342} C_VEL
LIN {X 0,Y 502.038,Z 500.356,A -85,B 0,C 180,E1 -5692.492,E2 -5692.492} C_VEL
LIN {X 0,Y 502.016,Z 500.192,A -85,B 0,C 180,E1 -5693.951,E2 -5693.951} C_VEL
LIN {X 0,Y 502.012,Z 499.483,A -85,B 0,C 180,E1 -5694.832,E2 -5694.832} C_VEL
LIN {X 0,Y 502.104,Z 497.038,A -85,B 0,C 180,E1 -5696.387,E2 -5696.387} C_VEL
LIN {X 0,Y 502.208,Z 493.335,A -85,B 0,C 180,E1 -5697.832,E2 -5697.832} C_VEL
LIN {X 0,Y 502.342,Z 488.002,A -85,B 0,C 180,E1 -5699.316,E2 -5699.316} C_VEL
LIN {X 0,Y 502.528,Z 481.378,A -85,B 0,C 180,E1 -5700.692,E2 -5700.692} C_VEL
LIN {X 0,Y 502.807,Z 473.981,A -85,B 0,C 180,E1 -5701.91,E2 -5701.91} C_VEL
LIN {X 0,Y 503.091,Z 465.401,A -85,B 0,C 180,E1 -5703.052,E2 -5703.052} C_VEL
LIN {X 0,Y 503.444,Z 455.07,A -85,B 0,C 180,E1 -5704.149,E2 -5704.149} C_VEL
LIN {X 0,Y 503.812,Z 445.1,A -85,B 0,C 180,E1 -5705.004,E2 -5705.004} C_VEL
LIN {X 0,Y 504.118,Z 434.884,A -85,B 0,C 180,E1 -5705.715,E2 -5705.715} C_VEL
LIN {X 0,Y 504.431,Z 423.472,A -85,B 0,C 180,E1 -5706.339,E2 -5706.339} C_VEL
LIN {X 0,Y 504.711,Z 411.053,A -85,B 0,C 180,E1 -5706.841,E2 -5706.841} C_VEL
LIN {X 0,Y 503.181,Z 402.378,A -85,B 0,C 180,E1 -5707.15,E2 -5707.15} C_VEL
LIN {X 0,Y 502.155,Z 398.015,A -85,B 0,C 180,E1 -5707.301,E2 -5707.301} C_VEL
LIN {X 0,Y 502.172,Z 394.975,A -85,B 0,C 180,E1 -5710.071,E2 -5710.071} C_VEL
LIN {X 0,Y 502.261,Z 391.494,A -85,B 0,C 180,E1 -5713.283,E2 -5713.283} C_VEL
LIN {X 0,Y 502.301,Z 389.01,A -85,B 0,C 180,E1 -5715.607,E2 -5715.607} C_VEL
LIN {X 0,Y 502.319,Z 385.492,A -85,B 0,C 180,E1 -5718.884,E2 -5718.884} C_VEL
LIN {X 0,Y 502.352,Z 382.14,A -85,B 0,C 180,E1 -5722.007,E2 -5722.007} C_VEL
LIN {X 0,Y 502.461,Z 378.909,A -85,B 0,C 180,E1 -5725.007,E2 -5725.007} C_VEL
LIN {X 0,Y 502.475,Z 377.9,A -85,B 0,C 180,E1 -5725.981,E2 -5725.981} C_VEL
LIN {X 0,Y 502.763,Z 377.861,A -85,B 0,C 180,E1 -5728.854,E2 -5728.854} C_VEL
LIN {X 0,Y 502.827,Z 377.851,A -85,B 0,C 180,E1 -5731.703,E2 -5731.703} C_VEL
LIN {X 0,Y 502.825,Z 377.852,A -85,B 0,C 180,E1 -5734.324,E2 -5734.324} C_VEL
LIN {X 0,Y 502.821,Z 377.853,A -85,B 0,C 180,E1 -5737.286,E2 -5737.286} C_VEL
LIN {X 0,Y 502.807,Z 377.856,A -85,B 0,C 180,E1 -5740.399,E2 -5740.399} C_VEL
LIN {X 0,Y 502.816,Z 377.854,A -85,B 0,C 180,E1 -5742.931,E2 -5742.931} C_VEL
LIN {X 0,Y 502.825,Z 377.851,A -85,B 0,C 180,E1 -5745.429,E2 -5745.429} C_VEL
LIN {X 0,Y 502.875,Z 377.847,A -85,B 0,C 180,E1 -5748.717,E2 -5748.717} C_VEL
LIN {X 0,Y 502.882,Z 377.844,A -85,B 0,C 180,E1 -5751.966,E2 -5751.966} C_VEL
LIN {X 0,Y 502.945,Z 377.837,A -85,B 0,C 180,E1 -5754.387,E2 -5754.387} C_VEL
LIN {X 0,Y 503.009,Z 377.828,A -85,B 0,C 180,E1 -5757.598,E2 -5757.598} C_VEL
LIN {X 0,Y 503.004,Z 377.829,A -85,B 0,C 180,E1 -5760,E2 -5760} C_VEL
LIN {X 0,Y 503.011,Z 377.829,A -85,B 0,C 180,E1 -5762.402,E2 -5762.402} C_VEL
LIN {X 0,Y 502.919,Z 377.839,A -85,B 0,C 180,E1 -5765.614,E2 -5765.614} C_VEL
LIN {X 0,Y 502.881,Z 377.844,A -85,B 0,C 180,E1 -5768.034,E2 -5768.034} C_VEL
LIN {X 0,Y 502.875,Z 377.846,A -85,B 0,C 180,E1 -5771.283,E2 -5771.283} C_VEL
LIN {X 0,Y 502.824,Z 377.853,A -85,B 0,C 180,E1 -5774.572,E2 -5774.572} C_VEL
LIN {X 0,Y 502.842,Z 377.85,A -85,B 0,C 180,E1 -5777.908,E2 -5777.908} C_VEL
LIN {X 0,Y 502.812,Z 377.853,A -85,B 0,C 180,E1 -5780.538,E2 -5780.538} C_VEL
LIN {X 0,Y 502.803,Z 377.855,A -85,B 0,C 180,E1 -5783.04,E2 -5783.04} C_VEL
LIN {X 0,Y 502.826,Z 377.852,A -85,B 0,C 180,E1 -5785.676,E2 -5785.676} C_VEL
LIN {X 0,Y 502.823,Z 377.853,A -85,B 0,C 180,E1 -5788.374,E2 -5788.374} C_VEL
LIN {X 0,Y 502.78,Z 377.859,A -85,B 0,C 180,E1 -5791.501,E2 -5791.501} C_VEL
LIN {X 0,Y 502.79,Z 377.859,A -85,B 0,C 180,E1 -5794.446,E2 -5794.446} C_VEL
LIN {X 0,Y 502.769,Z 377.861,A -85,B 0,C 180,E1 -5797.18,E2 -5797.18} C_VEL
LIN {X 0,Y 502.808,Z 377.858,A -85,B 0,C 180,E1 -5800.013,E2 -5800.013} C_VEL
LIN {X 0,Y 502.812,Z 377.856,A -85,B 0,C 180,E1 -5802.204,E2 -5802.204} C_VEL
LIN {X 0,Y 502.788,Z 377.863,A -85,B 0,C 180,E1 -5805.47,E2 -5805.47} C_VEL
LIN {X 0,Y 502.824,Z 377.857,A -85,B 0,C 180,E1 -5807.867,E2 -5807.867} C_VEL
LIN {X 0,Y 502.848,Z 378.01,A -85,B 0,C 180,E1 -5810.709,E2 -5810.709} C_VEL
LIN {X 0,Y 504.127,Z 385.117,A -85,B 0,C 180,E1 -5813.604,E2 -5813.604} C_VEL
LIN {X 0,Y 504.123,Z 390.672,A -85,B 0,C 180,E1 -5815.719,E2 -5815.719} C_VEL
LIN {X 0,Y 503.842,Z 397.924,A -85,B 0,C 180,E1 -5818.308,E2 -5818.308} C_VEL
LIN {X 0,Y 503.53,Z 407.913,A -85,B 0,C 180,E1 -5821.672,E2 -5821.672} C_VEL
LIN {X 0,Y 503.294,Z 416.021,A -85,B 0,C 180,E1 -5824.352,E2 -5824.352} C_VEL
LIN {X 0,Y 503.062,Z 425.004,A -85,B 0,C 180,E1 -5827.228,E2 -5827.228} C_VEL
LIN {X 0,Y 502.869,Z 433.498,A -85,B 0,C 180,E1 -5829.978,E2 -5829.978} C_VEL
LIN {X 0,Y 502.624,Z 442.766,A -85,B 0,C 180,E1 -5832.926,E2 -5832.926} C_VEL
LIN {X 0,Y 502.497,Z 451.578,A -85,B 0,C 180,E1 -5835.692,E2 -5835.692} C_VEL
LIN {X 0,Y 504.702,Z 465.16,A -85,B 0,C 180,E1 -5836.077,E2 -5836.077} C_VEL
LIN {X 0,Y 504.424,Z 478.153,A -85,B 0,C 180,E1 -5836.557,E2 -5836.557} C_VEL
LIN {X 0,Y 504.036,Z 490.59,A -85,B 0,C 180,E1 -5837.191,E2 -5837.191} C_VEL
LIN {X 0,Y 503.739,Z 501.613,A -85,B 0,C 180,E1 -5837.922,E2 -5837.922} C_VEL
LIN {X 0,Y 503.381,Z 512.488,A -85,B 0,C 180,E1 -5838.832,E2 -5838.832} C_VEL
LIN {X 0,Y 503.023,Z 521.349,A -85,B 0,C 180,E1 -5839.741,E2 -5839.741} C_VEL
LIN {X 0,Y 502.703,Z 530.973,A -85,B 0,C 180,E1 -5840.953,E2 -5840.953} C_VEL
LIN {X 0,Y 502.469,Z 538.631,A -85,B 0,C 180,E1 -5842.164,E2 -5842.164} C_VEL
LIN {X 0,Y 502.274,Z 545.687,A -85,B 0,C 180,E1 -5843.575,E2 -5843.575} C_VEL
LIN {X 0,Y 502.185,Z 550.378,A -85,B 0,C 180,E1 -5844.782,E2 -5844.782} C_VEL
LIN {X 0,Y 502.151,Z 553.962,A -85,B 0,C 180,E1 -5845.989,E2 -5845.989} C_VEL
LIN {X 0,Y 502.12,Z 555.811,A -85,B 0,C 180,E1 -5846.792,E2 -5846.792} C_VEL
LIN {X 0,Y 502.066,Z 557.198,A -85,B 0,C 180,E1 -5847.595,E2 -5847.595} C_VEL
LIN {X 0,Y 501.99,Z 558.787,A -85,B 0,C 180,E1 -5849.199,E2 -5849.199} C_VEL
LIN {X 0,Y 501.98,Z 559,A -85,B 0,C 180,E1 -5850.002,E2 -5850.002} C_VEL
LIN {X 0,Y 502.036,Z 558.183,A -85,B 0,C 180,E1 -5851.606,E2 -5851.606} C_VEL
LIN {X 0,Y 502.066,Z 557.195,A -85,B 0,C 180,E1 -5852.408,E2 -5852.408} C_VEL
LIN {X 0,Y 502.121,Z 555.807,A -85,B 0,C 180,E1 -5853.211,E2 -5853.211} C_VEL
LIN {X 0,Y 502.129,Z 552.891,A -85,B 0,C 180,E1 -5854.416,E2 -5854.416} C_VEL
LIN {X 0,Y 502.261,Z 548.943,A -85,B 0,C 180,E1 -5855.623,E2 -5855.623} C_VEL
LIN {X 0,Y 502.337,Z 542.97,A -85,B 0,C 180,E1 -5857.013,E2 -5857.013} C_VEL
LIN {X 0,Y 502.543,Z 536.228,A -85,B 0,C 180,E1 -5858.243,E2 -5858.243} C_VEL
LIN {X 0,Y 502.812,Z 527.981,A -85,B 0,C 180,E1 -5859.454,E2 -5859.454} C_VEL
LIN {X 0,Y 503.072,Z 519.527,A -85,B 0,C 180,E1 -5860.465,E2 -5860.465} C_VEL
LIN {X 0,Y 503.5,Z 509.079,A -85,B 0,C 180,E1 -5861.474,E2 -5861.474} C_VEL
LIN {X 0,Y 503.796,Z 497.409,A -85,B 0,C 180,E1 -5862.379,E2 -5862.379} C_VEL
LIN {X 0,Y 504.151,Z 485.464,A -85,B 0,C 180,E1 -5863.094,E2 -5863.094} C_VEL
LIN {X 0,Y 504.523,Z 473.134,A -85,B 0,C 180,E1 -5863.648,E2 -5863.648} C_VEL
LIN {X 0,Y 504.524,Z 464.129,A -85,B 0,C 180,E1 -5863.956,E2 -5863.956} C_VEL
LIN {X 0,Y 502.491,Z 451.526,A -85,B 0,C 180,E1 -5864.324,E2 -5864.324} C_VEL
LIN {X 0,Y 502.666,Z 441.432,A -85,B 0,C 180,E1 -5867.495,E2 -5867.495} C_VEL
LIN {X 0,Y 502.907,Z 431.827,A -85,B 0,C 180,E1 -5870.559,E2 -5870.559} C_VEL
LIN {X 0,Y 503.13,Z 422.897,A -85,B 0,C 180,E1 -5873.461,E2 -5873.461} C_VEL
LIN {X 0,Y 503.403,Z 413.332,A -85,B 0,C 180,E1 -5876.537,E2 -5876.537} C_VEL
LIN {X 0,Y 503.658,Z 404.123,A -85,B 0,C 180,E1 -5879.675,E2 -5879.675} C_VEL
LIN {X 0,Y 504.026,Z 394.729,A -85,B 0,C 180,E1 -5882.944,E2 -5882.944} C_VEL
LIN {X 0,Y 504.267,Z 387.995,A -85,B 0,C 180,E1 -5885.338,E2 -5885.338} C_VEL
LIN {X 0,Y 503.943,Z 384.038,A -85,B 0,C 180,E1 -5886.848,E2 -5886.848} C_VEL
LIN {X 0,Y 502.81,Z 377.857,A -85,B 0,C 180,E1 -5889.428,E2 -5889.428} C_VEL
LIN {X 0,Y 502.809,Z 377.856,A -85,B 0,C 180,E1 -5892.2,E2 -5892.2} C_VEL
LIN {X 0,Y 502.791,Z 377.859,A -85,B 0,C 180,E1 -5895.47,E2 -5895.47} C_VEL
LIN {X 0,Y 502.825,Z 377.853,A -85,B 0,C 180,E1 -5898.934,E2 -5898.934} C_VEL
LIN {X 0,Y 502.798,Z 377.856,A -85,B 0,C 180,E1 -5902.046,E2 -5902.046} C_VEL
LIN {X 0,Y 502.8,Z 377.856,A -85,B 0,C 180,E1 -5905.034,E2 -5905.034} C_VEL
LIN {X 0,Y 502.787,Z 377.857,A -85,B 0,C 180,E1 -5907.915,E2 -5907.915} C_VEL
LIN {X 0,Y 502.829,Z 377.853,A -85,B 0,C 180,E1 -5910.712,E2 -5910.712} C_VEL
LIN {X 0,Y 502.868,Z 377.846,A -85,B 0,C 180,E1 -5913.439,E2 -5913.439} C_VEL
LIN {X 0,Y 502.79,Z 377.857,A -85,B 0,C 180,E1 -5916.086,E2 -5916.086} C_VEL
LIN {X 0,Y 502.788,Z 377.858,A -85,B 0,C 180,E1 -5918.689,E2 -5918.689} C_VEL
LIN {X 0,Y 502.835,Z 377.852,A -85,B 0,C 180,E1 -5921.248,E2 -5921.248} C_VEL
LIN {X 0,Y 502.826,Z 377.853,A -85,B 0,C 180,E1 -5923.767,E2 -5923.767} C_VEL
LIN {X 0,Y 502.835,Z 377.852,A -85,B 0,C 180,E1 -5926.255,E2 -5926.255} C_VEL
LIN {X 0,Y 502.881,Z 377.846,A -85,B 0,C 180,E1 -5928.717,E2 -5928.717} C_VEL
LIN {X 0,Y 502.906,Z 377.844,A -85,B 0,C 180,E1 -5931.967,E2 -5931.967} C_VEL
LIN {X 0,Y 502.938,Z 377.839,A -85,B 0,C 180,E1 -5934.386,E2 -5934.386} C_VEL
LIN {X 0,Y 503.028,Z 377.827,A -85,B 0,C 180,E1 -5937.598,E2 -5937.598} C_VEL
LIN {X 0,Y 503.031,Z 377.829,A -85,B 0,C 180,E1 -5940,E2 -5940} C_VEL
LIN {X 0,Y 503.027,Z 377.828,A -85,B 0,C 180,E1 -5942.402,E2 -5942.402} C_VEL
LIN {X 0,Y 502.937,Z 377.839,A -85,B 0,C 180,E1 -5945.613,E2 -5945.613} C_VEL
LIN {X 0,Y 502.906,Z 377.843,A -85,B 0,C 180,E1 -5948.033,E2 -5948.033} C_VEL
LIN {X 0,Y 502.881,Z 377.845,A -85,B 0,C 180,E1 -5951.283,E2 -5951.283} C_VEL
LIN {X 0,Y 502.849,Z 377.85,A -85,B 0,C 180,E1 -5954.571,E2 -5954.571} C_VEL
LIN {X 0,Y 502.859,Z 377.849,A -85,B 0,C 180,E1 -5957.907,E2 -5957.907} C_VEL
LIN {X 0,Y 502.834,Z 377.852,A -85,B 0,C 180,E1 -5960.536,E2 -5960.536} C_VEL
LIN {X 0,Y 502.795,Z 377.857,A -85,B 0,C 180,E1 -5963.04,E2 -5963.04} C_VEL
LIN {X 0,Y 502.844,Z 377.851,A -85,B 0,C 180,E1 -5965.675,E2 -5965.675} C_VEL
LIN {X 0,Y 502.845,Z 377.849,A -85,B 0,C 180,E1 -5968.372,E2 -5968.372} C_VEL
LIN {X 0,Y 502.797,Z 377.857,A -85,B 0,C 180,E1 -5971.498,E2 -5971.498} C_VEL
LIN {X 0,Y 502.808,Z 377.856,A -85,B 0,C 180,E1 -5973.994,E2 -5973.994} C_VEL
LIN {X 0,Y 502.781,Z 377.859,A -85,B 0,C 180,E1 -5977.177,E2 -5977.177} C_VEL
LIN {X 0,Y 502.792,Z 377.856,A -85,B 0,C 180,E1 -5980.015,E2 -5980.015} C_VEL
LIN {X 0,Y 502.808,Z 377.854,A -85,B 0,C 180,E1 -5982.199,E2 -5982.199} C_VEL
LIN {X 0,Y 502.791,Z 377.858,A -85,B 0,C 180,E1 -5985.47,E2 -5985.47} C_VEL
LIN {X 0,Y 502.825,Z 377.854,A -85,B 0,C 180,E1 -5988.934,E2 -5988.934} C_VEL
LIN {X 0,Y 502.798,Z 377.856,A -85,B 0,C 180,E1 -5992.045,E2 -5992.045} C_VEL
LIN {X 0,Y 502.804,Z 377.857,A -85,B 0,C 180,E1 -5995.034,E2 -5995.034} C_VEL
LIN {X 0,Y 502.813,Z 377.854,A -85,B 0,C 180,E1 -5997.223,E2 -5997.223} C_VEL
LIN {X 0,Y 502.111,Z 377.941,A -85,B 0,C 180,E1 -5997.892,E2 -5997.892} C_VEL
LIN {X 0,Y 499.246,Z 378.3,A -85,B 0,C 180,E1 -5998.978,E2 -5998.978} C_VEL
LIN {X 0,Y 496.852,Z 378.597,A -85,B 0,C 180,E1 -5999.853,E2 -5999.853} C_VEL
LIN {X 0,Y 495.836,Z 378.724,A -85,B 0,C 180,E1 -6000.528,E2 -6000.528} C_VEL
LIN {X 0,Y 495.758,Z 378.732,A -85,B 0,C 180,E1 -6000.757,E2 -6000.757} C_VEL
LIN {X 0,Y 495.796,Z 378.726,A -85,B 0,C 180,E1 -6003.931,E2 -6003.931} C_VEL
LIN {X 0,Y 495.765,Z 378.733,A -85,B 0,C 180,E1 -6007.138,E2 -6007.138} C_VEL
LIN {X 0,Y 495.776,Z 378.73,A -85,B 0,C 180,E1 -6010.109,E2 -6010.109} C_VEL
LIN {X 0,Y 495.786,Z 378.731,A -85,B 0,C 180,E1 -6012.68,E2 -6012.68} C_VEL
LIN {X 0,Y 495.794,Z 378.728,A -85,B 0,C 180,E1 -6015.216,E2 -6015.216} C_VEL
LIN {X 0,Y 495.788,Z 378.73,A -85,B 0,C 180,E1 -6017.988,E2 -6017.988} C_VEL
LIN {X 0,Y 495.469,Z 378.771,A -85,B 0,C 180,E1 -6020.198,E2 -6020.198} C_VEL
LIN {X 0,Y 495.425,Z 379.047,A -85,B 0,C 180,E1 -6021.021,E2 -6021.021} C_VEL
LIN {X 0,Y 495.419,Z 381.668,A -85,B 0,C 180,E1 -6023.482,E2 -6023.482} C_VEL
LIN {X 0,Y 495.427,Z 384.287,A -85,B 0,C 180,E1 -6025.931,E2 -6025.931} C_VEL
LIN {X 0,Y 495.215,Z 388.73,A -85,B 0,C 180,E1 -6029.998,E2 -6029.998} C_VEL
LIN {X 0,Y 495.229,Z 393.152,A -85,B 0,C 180,E1 -6034.067,E2 -6034.067} C_VEL
LIN {X 0,Y 495.202,Z 395.93,A -85,B 0,C 180,E1 -6036.559,E2 -6036.559} C_VEL
LIN {X 0,Y 495.1,Z 398.264,A -85,B 0,C 180,E1 -6038.596,E2 -6038.596} C_VEL
LIN {X 0,Y 497.633,Z 410.227,A -85,B 0,C 180,E1 -6039.012,E2 -6039.012} C_VEL
LIN {X 0,Y 497.642,Z 421.154,A -85,B 0,C 180,E1 -6039.448,E2 -6039.448} C_VEL
LIN {X 0,Y 497.225,Z 433.131,A -85,B 0,C 180,E1 -6040.072,E2 -6040.072} C_VEL
LIN {X 0,Y 496.879,Z 443.924,A -85,B 0,C 180,E1 -6040.8,E2 -6040.8} C_VEL
LIN {X 0,Y 496.52,Z 454.791,A -85,B 0,C 180,E1 -6041.728,E2 -6041.728} C_VEL
LIN {X 0,Y 496.171,Z 463.508,A -85,B 0,C 180,E1 -6042.639,E2 -6042.639} C_VEL
LIN {X 0,Y 495.842,Z 472.101,A -85,B 0,C 180,E1 -6043.732,E2 -6043.732} C_VEL
LIN {X 0,Y 495.606,Z 478.912,A -85,B 0,C 180,E1 -6044.787,E2 -6044.787} C_VEL
LIN {X 0,Y 495.39,Z 485.609,A -85,B 0,C 180,E1 -6046.058,E2 -6046.058} C_VEL
LIN {X 0,Y 495.228,Z 490.904,A -85,B 0,C 180,E1 -6047.337,E2 -6047.337} C_VEL
LIN {X 0,Y 495.11,Z 494.984,A -85,B 0,C 180,E1 -6048.624,E2 -6048.624} C_VEL
LIN {X 0,Y 494.979,Z 498.855,A -85,B 0,C 180,E1 -6050.429,E2 -6050.429} C_VEL
LIN {X 0,Y 494.953,Z 500.319,A -85,B 0,C 180,E1 -6051.663,E2 -6051.663} C_VEL
LIN {X 0,Y 494.973,Z 500.818,A -85,B 0,C 180,E1 -6052.643,E2 -6052.643} C_VEL
LIN {X 0,Y 494.957,Z 500.422,A -85,B 0,C 180,E1 -6054.314,E2 -6054.314} C_VEL
LIN {X 0,Y 494.942,Z 499.496,A -85,B 0,C 180,E1 -6055.211,E2 -6055.211} C_VEL
LIN {X 0,Y 495.032,Z 497.188,A -85,B 0,C 180,E1 -6056.566,E2 -6056.566} C_VEL
LIN {X 0,Y 495.161,Z 493.69,A -85,B 0,C 180,E1 -6057.927,E2 -6057.927} C_VEL
LIN {X 0,Y 495.294,Z 488.826,A -85,B 0,C 180,E1 -6059.308,E2 -6059.308} C_VEL
LIN {X 0,Y 495.489,Z 482.345,A -85,B 0,C 180,E1 -6060.703,E2 -6060.703} C_VEL
LIN {X 0,Y 495.825,Z 474.25,A -85,B 0,C 180,E1 -6062.061,E2 -6062.061} C_VEL
LIN {X 0,Y 496.137,Z 465.575,A -85,B 0,C 180,E1 -6063.224,E2 -6063.224} C_VEL
LIN {X 0,Y 496.479,Z 456.199,A -85,B 0,C 180,E1 -6064.239,E2 -6064.239} C_VEL
LIN {X 0,Y 496.886,Z 445.445,A -85,B 0,C 180,E1 -6065.181,E2 -6065.181} C_VEL
LIN {X 0,Y 497.267,Z 434.07,A -85,B 0,C 180,E1 -6065.971,E2 -6065.971} C_VEL
LIN {X 0,Y 497.597,Z 422.653,A -85,B 0,C 180,E1 -6066.583,E2 -6066.583} C_VEL
LIN {X 0,Y 497.699,Z 410.413,A -85,B 0,C 180,E1 -6067.076,E2 -6067.076} C_VEL
LIN {X 0,Y 495.254,Z 399.518,A -85,B 0,C 180,E1 -6067.458,E2 -6067.458} C_VEL
LIN {X 0,Y 495.072,Z 398.445,A -85,B 0,C 180,E1 -6067.514,E2 -6067.514} C_VEL
LIN {X 0,Y 495.114,Z 394.92,A -85,B 0,C 180,E1 -6070.762,E2 -6070.762} C_VEL
LIN {X 0,Y 495.18,Z 391.815,A -85,B 0,C 180,E1 -6073.628,E2 -6073.628} C_VEL
LIN {X 0,Y 495.223,Z 388.906,A -85,B 0,C 180,E1 -6076.363,E2 -6076.363} C_VEL
LIN {X 0,Y 495.276,Z 385.828,A -85,B 0,C 180,E1 -6079.251,E2 -6079.251} C_VEL
LIN {X 0,Y 495.332,Z 382.252,A -85,B 0,C 180,E1 -6082.609,E2 -6082.609} C_VEL
LIN {X 0,Y 495.429,Z 379.241,A -85,B 0,C 180,E1 -6085.429,E2 -6085.429} C_VEL
LIN {X 0,Y 495.528,Z 378.765,A -85,B 0,C 180,E1 -6086.798,E2 -6086.798} C_VEL
LIN {X 0,Y 495.729,Z 378.738,A -85,B 0,C 180,E1 -6089.311,E2 -6089.311} C_VEL
LIN {X 0,Y 495.765,Z 378.732,A -85,B 0,C 180,E1 -6092.108,E2 -6092.108} C_VEL
LIN {X 0,Y 495.774,Z 378.732,A -85,B 0,C 180,E1 -6094.832,E2 -6094.832} C_VEL
LIN {X 0,Y 495.765,Z 378.733,A -85,B 0,C 180,E1 -6097.496,E2 -6097.496} C_VEL
LIN {X 0,Y 495.759,Z 378.731,A -85,B 0,C 180,E1 -6100.109,E2 -6100.109} C_VEL
LIN {X 0,Y 495.768,Z 378.73,A -85,B 0,C 180,E1 -6102.681,E2 -6102.681} C_VEL
LIN {X 0,Y 495.77,Z 378.73,A -85,B 0,C 180,E1 -6105.217,E2 -6105.217} C_VEL
LIN {X 0,Y 495.849,Z 378.724,A -85,B 0,C 180,E1 -6108.555,E2 -6108.555} C_VEL
LIN {X 0,Y 495.853,Z 378.719,A -85,B 0,C 180,E1 -6111.852,E2 -6111.852} C_VEL
LIN {X 0,Y 495.899,Z 378.715,A -85,B 0,C 180,E1 -6114.307,E2 -6114.307} C_VEL
LIN {X 0,Y 495.977,Z 378.704,A -85,B 0,C 180,E1 -6117.564,E2 -6117.564} C_VEL
LIN {X 0,Y 495.975,Z 378.704,A -85,B 0,C 180,E1 -6120,E2 -6120} C_VEL
LIN {X 0,Y 495.98,Z 378.705,A -85,B 0,C 180,E1 -6122.436,E2 -6122.436} C_VEL
LIN {X 0,Y 495.877,Z 378.717,A -85,B 0,C 180,E1 -6125.694,E2 -6125.694} C_VEL
LIN {X 0,Y 495.852,Z 378.72,A -85,B 0,C 180,E1 -6128.148,E2 -6128.148} C_VEL
LIN {X 0,Y 495.849,Z 378.722,A -85,B 0,C 180,E1 -6131.445,E2 -6131.445} C_VEL
LIN {X 0,Y 495.769,Z 378.73,A -85,B 0,C 180,E1 -6134.784,E2 -6134.784} C_VEL
LIN {X 0,Y 495.769,Z 378.731,A -85,B 0,C 180,E1 -6137.319,E2 -6137.319} C_VEL
LIN {X 0,Y 495.76,Z 378.734,A -85,B 0,C 180,E1 -6139.891,E2 -6139.891} C_VEL
LIN {X 0,Y 495.771,Z 378.731,A -85,B 0,C 180,E1 -6142.87,E2 -6142.87} C_VEL
LIN {X 0,Y 495.783,Z 378.731,A -85,B 0,C 180,E1 -6146.068,E2 -6146.068} C_VEL
LIN {X 0,Y 495.755,Z 378.735,A -85,B 0,C 180,E1 -6148.816,E2 -6148.816} C_VEL
LIN {X 0,Y 495.742,Z 378.737,A -85,B 0,C 180,E1 -6151.727,E2 -6151.727} C_VEL
LIN {X 0,Y 495.76,Z 378.734,A -85,B 0,C 180,E1 -6154.697,E2 -6154.697} C_VEL
LIN {X 0,Y 495.719,Z 378.738,A -85,B 0,C 180,E1 -6157.563,E2 -6157.563} C_VEL
LIN {X 0,Y 495.767,Z 378.733,A -85,B 0,C 180,E1 -6160.7,E2 -6160.7} C_VEL
LIN {X 0,Y 495.721,Z 378.742,A -85,B 0,C 180,E1 -6163.697,E2 -6163.697} C_VEL
LIN {X 0,Y 495.723,Z 378.742,A -85,B 0,C 180,E1 -6166.306,E2 -6166.306} C_VEL
LIN {X 0,Y 495.771,Z 378.734,A -85,B 0,C 180,E1 -6169.304,E2 -6169.304} C_VEL
LIN {X 0,Y 495.783,Z 378.739,A -85,B 0,C 180,E1 -6170.368,E2 -6170.368} C_VEL
LIN {X 0,Y 497.184,Z 386.648,A -85,B 0,C 180,E1 -6173.681,E2 -6173.681} C_VEL
LIN {X 0,Y 497.189,Z 391.692,A -85,B 0,C 180,E1 -6175.571,E2 -6175.571} C_VEL
LIN {X 0,Y 496.802,Z 399.498,A -85,B 0,C 180,E1 -6178.441,E2 -6178.441} C_VEL
LIN {X 0,Y 496.513,Z 409.196,A -85,B 0,C 180,E1 -6181.752,E2 -6181.752} C_VEL
LIN {X 0,Y 496.247,Z 417.06,A -85,B 0,C 180,E1 -6184.411,E2 -6184.411} C_VEL
LIN {X 0,Y 496.016,Z 426.825,A -85,B 0,C 180,E1 -6187.51,E2 -6187.51} C_VEL
LIN {X 0,Y 495.769,Z 436.146,A -85,B 0,C 180,E1 -6190.543,E2 -6190.543} C_VEL
LIN {X 0,Y 495.546,Z 445.413,A -85,B 0,C 180,E1 -6193.524,E2 -6193.524} C_VEL
LIN {X 0,Y 495.446,Z 451.649,A -85,B 0,C 180,E1 -6195.487,E2 -6195.487} C_VEL
LIN {X 0,Y 497.679,Z 465.16,A -85,B 0,C 180,E1 -6195.877,E2 -6195.877} C_VEL
LIN {X 0,Y 497.534,Z 478.152,A -85,B 0,C 180,E1 -6196.368,E2 -6196.368} C_VEL
LIN {X 0,Y 497.107,Z 490.725,A -85,B 0,C 180,E1 -6197.018,E2 -6197.018} C_VEL
LIN {X 0,Y 496.783,Z 501.613,A -85,B 0,C 180,E1 -6197.75,E2 -6197.75} C_VEL
LIN {X 0,Y 496.407,Z 512.487,A -85,B 0,C 180,E1 -6198.673,E2 -6198.673} C_VEL
LIN {X 0,Y 495.996,Z 521.349,A -85,B 0,C 180,E1 -6199.594,E2 -6199.594} C_VEL
LIN {X 0,Y 495.671,Z 530.973,A -85,B 0,C 180,E1 -6200.823,E2 -6200.823} C_VEL
LIN {X 0,Y 495.402,Z 538.631,A -85,B 0,C 180,E1 -6202.051,E2 -6202.051} C_VEL
LIN {X 0,Y 495.202,Z 545.687,A -85,B 0,C 180,E1 -6203.482,E2 -6203.482} C_VEL
LIN {X 0,Y 495.122,Z 550.379,A -85,B 0,C 180,E1 -6204.708,E2 -6204.708} C_VEL
LIN {X 0,Y 495.049,Z 553.963,A -85,B 0,C 180,E1 -6205.931,E2 -6205.931} C_VEL
LIN {X 0,Y 495.042,Z 555.81,A -85,B 0,C 180,E1 -6206.746,E2 -6206.746} C_VEL
LIN {X 0,Y 494.961,Z 558.185,A -85,B 0,C 180,E1 -6208.374,E2 -6208.374} C_VEL
LIN {X 0,Y 494.898,Z 559,A -85,B 0,C 180,E1 -6210.002,E2 -6210.002} C_VEL
LIN {X 0,Y 494.961,Z 558.183,A -85,B 0,C 180,E1 -6211.629,E2 -6211.629} C_VEL
LIN {X 0,Y 495.043,Z 555.807,A -85,B 0,C 180,E1 -6213.257,E2 -6213.257} C_VEL
LIN {X 0,Y 495.029,Z 552.891,A -85,B 0,C 180,E1 -6214.48,E2 -6214.48} C_VEL
LIN {X 0,Y 495.211,Z 547.797,A -85,B 0,C 180,E1 -6216,E2 -6216} C_VEL
LIN {X 0,Y 495.279,Z 541.862,A -85,B 0,C 180,E1 -6217.339,E2 -6217.339} C_VEL
LIN {X 0,Y 495.558,Z 534.994,A -85,B 0,C 180,E1 -6218.565,E2 -6218.565} C_VEL
LIN {X 0,Y 495.853,Z 526.402,A -85,B 0,C 180,E1 -6219.794,E2 -6219.794} C_VEL
LIN {X 0,Y 496.21,Z 517.586,A -85,B 0,C 180,E1 -6220.818,E2 -6220.818} C_VEL
LIN {X 0,Y 496.605,Z 506.729,A -85,B 0,C 180,E1 -6221.843,E2 -6221.843} C_VEL
LIN {X 0,Y 496.901,Z 496.191,A -85,B 0,C 180,E1 -6222.637,E2 -6222.637} C_VEL
LIN {X 0,Y 497.324,Z 483.475,A -85,B 0,C 180,E1 -6223.381,E2 -6223.381} C_VEL
LIN {X 0,Y 497.709,Z 470.453,A -85,B 0,C 180,E1 -6223.943,E2 -6223.943} C_VEL
LIN {X 0,Y 497.542,Z 464.128,A -85,B 0,C 180,E1 -6224.156,E2 -6224.156} C_VEL
LIN {X 0,Y 495.431,Z 451.526,A -85,B 0,C 180,E1 -6224.533,E2 -6224.533} C_VEL
LIN {X 0,Y 495.642,Z 441.432,A -85,B 0,C 180,E1 -6227.751,E2 -6227.751} C_VEL
LIN {X 0,Y 495.889,Z 432.164,A -85,B 0,C 180,E1 -6230.753,E2 -6230.753} C_VEL
LIN {X 0,Y 496.107,Z 422.669,A -85,B 0,C 180,E1 -6233.813,E2 -6233.813} C_VEL
LIN {X 0,Y 496.344,Z 414.544,A -85,B 0,C 180,E1 -6236.455,E2 -6236.455} C_VEL
LIN {X 0,Y 496.638,Z 405.18,A -85,B 0,C 180,E1 -6239.69,E2 -6239.69} C_VEL
LIN {X 0,Y 497.036,Z 395.87,A -85,B 0,C 180,E1 -6242.984,E2 -6242.984} C_VEL
LIN {X 0,Y 497.31,Z 389.187,A -85,B 0,C 180,E1 -6245.41,E2 -6245.41} C_VEL
LIN {X 0,Y 496.956,Z 385.259,A -85,B 0,C 180,E1 -6246.945,E2 -6246.945} C_VEL
LIN {X 0,Y 495.77,Z 378.733,A -85,B 0,C 180,E1 -6249.74,E2 -6249.74} C_VEL
LIN {X 0,Y 495.731,Z 378.737,A -85,B 0,C 180,E1 -6252.884,E2 -6252.884} C_VEL
LIN {X 0,Y 495.733,Z 378.737,A -85,B 0,C 180,E1 -6255.999,E2 -6255.999} C_VEL
LIN {X 0,Y 495.772,Z 378.732,A -85,B 0,C 180,E1 -6259.3,E2 -6259.3} C_VEL
LIN {X 0,Y 495.734,Z 378.736,A -85,B 0,C 180,E1 -6262.439,E2 -6262.439} C_VEL
LIN {X 0,Y 495.776,Z 378.73,A -85,B 0,C 180,E1 -6265.456,E2 -6265.456} C_VEL
LIN {X 0,Y 495.76,Z 378.733,A -85,B 0,C 180,E1 -6268.364,E2 -6268.364} C_VEL
LIN {X 0,Y 495.792,Z 378.727,A -85,B 0,C 180,E1 -6271.507,E2 -6271.507} C_VEL
LIN {X 0,Y 495.795,Z 378.727,A -85,B 0,C 180,E1 -6273.932,E2 -6273.932} C_VEL
LIN {X 0,Y 495.765,Z 378.733,A -85,B 0,C 180,E1 -6277.139,E2 -6277.139} C_VEL
LIN {X 0,Y 495.776,Z 378.731,A -85,B 0,C 180,E1 -6280.11,E2 -6280.11} C_VEL
LIN {X 0,Y 495.791,Z 378.729,A -85,B 0,C 180,E1 -6282.681,E2 -6282.681} C_VEL
LIN {X 0,Y 495.795,Z 378.728,A -85,B 0,C 180,E1 -6285.217,E2 -6285.217} C_VEL
LIN {X 0,Y 495.856,Z 378.723,A -85,B 0,C 180,E1 -6288.555,E2 -6288.555} C_VEL
LIN {X 0,Y 495.878,Z 378.719,A -85,B 0,C 180,E1 -6291.852,E2 -6291.852} C_VEL
LIN {X 0,Y 495.895,Z 378.716,A -85,B 0,C 180,E1 -6294.306,E2 -6294.306} C_VEL
LIN {X 0,Y 495.996,Z 378.703,A -85,B 0,C 180,E1 -6297.564,E2 -6297.564} C_VEL
LIN {X 0,Y 495.986,Z 378.705,A -85,B 0,C 180,E1 -6300.812,E2 -6300.812} C_VEL
LIN {X 0,Y 495.996,Z 378.703,A -85,B 0,C 180,E1 -6302.436,E2 -6302.436} C_VEL
LIN {X 0,Y 495.893,Z 378.717,A -85,B 0,C 180,E1 -6305.693,E2 -6305.693} C_VEL
LIN {X 0,Y 495.878,Z 378.719,A -85,B 0,C 180,E1 -6308.148,E2 -6308.148} C_VEL
LIN {X 0,Y 495.856,Z 378.721,A -85,B 0,C 180,E1 -6311.445,E2 -6311.445} C_VEL
LIN {X 0,Y 495.794,Z 378.728,A -85,B 0,C 180,E1 -6314.783,E2 -6314.783} C_VEL
LIN {X 0,Y 495.785,Z 378.729,A -85,B 0,C 180,E1 -6317.319,E2 -6317.319} C_VEL
LIN {X 0,Y 495.775,Z 378.732,A -85,B 0,C 180,E1 -6319.89,E2 -6319.89} C_VEL
LIN {X 0,Y 495.764,Z 378.732,A -85,B 0,C 180,E1 -6322.86,E2 -6322.86} C_VEL
LIN {X 0,Y 495.795,Z 378.728,A -85,B 0,C 180,E1 -6326.068,E2 -6326.068} C_VEL
LIN {X 0,Y 495.776,Z 378.729,A -85,B 0,C 180,E1 -6328.814,E2 -6328.814} C_VEL
LIN {X 0,Y 495.76,Z 378.733,A -85,B 0,C 180,E1 -6331.725,E2 -6331.725} C_VEL
LIN {X 0,Y 495.773,Z 378.731,A -85,B 0,C 180,E1 -6334.693,E2 -6334.693} C_VEL
LIN {X 0,Y 495.733,Z 378.737,A -85,B 0,C 180,E1 -6337.561,E2 -6337.561} C_VEL
LIN {X 0,Y 495.771,Z 378.732,A -85,B 0,C 180,E1 -6340.7,E2 -6340.7} C_VEL
LIN {X 0,Y 495.732,Z 378.735,A -85,B 0,C 180,E1 -6344.001,E2 -6344.001} C_VEL
LIN {X 0,Y 495.731,Z 378.737,A -85,B 0,C 180,E1 -6347.116,E2 -6347.116} C_VEL
LIN {X 0,Y 495.764,Z 378.732,A -85,B 0,C 180,E1 -6349.952,E2 -6349.952} C_VEL
LIN {X 0,Y 495.733,Z 378.736,A -85,B 0,C 180,E1 -6352.553,E2 -6352.553} C_VEL
LIN {X 0,Y 495.783,Z 378.73,A -85,B 0,C 180,E1 -6355.456,E2 -6355.456} C_VEL
LIN {X 0,Y 495.76,Z 378.734,A -85,B 0,C 180,E1 -6358.363,E2 -6358.363} C_VEL
LIN {X 0,Y 495.758,Z 378.732,A -85,B 0,C 180,E1 -6360.757,E2 -6360.757} C_VEL
LIN {X 0,Y 495.1,Z 378.816,A -85,B 0,C 180,E1 -6361.436,E2 -6361.436} C_VEL
LIN {X 0,Y 492.244,Z 379.172,A -85,B 0,C 180,E1 -6362.539,E2 -6362.539} C_VEL
LIN {X 0,Y 489.836,Z 379.47,A -85,B 0,C 180,E1 -6363.427,E2 -6363.427} C_VEL
LIN {X 0,Y 488.82,Z 379.596,A -85,B 0,C 180,E1 -6364.114,E2 -6364.114} C_VEL
LIN {X 0,Y 488.748,Z 379.606,A -85,B 0,C 180,E1 -6364.346,E2 -6364.346} C_VEL
LIN {X 0,Y 488.728,Z 379.61,A -85,B 0,C 180,E1 -6367.152,E2 -6367.152} C_VEL
LIN {X 0,Y 488.73,Z 379.608,A -85,B 0,C 180,E1 -6369.809,E2 -6369.809} C_VEL
LIN {X 0,Y 488.734,Z 379.609,A -85,B 0,C 180,E1 -6372.422,E2 -6372.422} C_VEL
LIN {X 0,Y 488.766,Z 379.604,A -85,B 0,C 180,E1 -6374.998,E2 -6374.998} C_VEL
LIN {X 0,Y 488.715,Z 379.612,A -85,B 0,C 180,E1 -6378.384,E2 -6378.384} C_VEL
LIN {X 0,Y 488.367,Z 379.657,A -85,B 0,C 180,E1 -6380.89,E2 -6380.89} C_VEL
LIN {X 0,Y 488.359,Z 382.267,A -85,B 0,C 180,E1 -6383.388,E2 -6383.388} C_VEL
LIN {X 0,Y 488.383,Z 384.91,A -85,B 0,C 180,E1 -6385.872,E2 -6385.872} C_VEL
LIN {X 0,Y 488.144,Z 389.398,A -85,B 0,C 180,E1 -6389.998,E2 -6389.998} C_VEL
LIN {X 0,Y 488.154,Z 392.987,A -85,B 0,C 180,E1 -6393.3,E2 -6393.3} C_VEL
LIN {X 0,Y 488.136,Z 396.572,A -85,B 0,C 180,E1 -6396.612,E2 -6396.612} C_VEL
LIN {X 0,Y 488.041,Z 398.655,A -85,B 0,C 180,E1 -6398.389,E2 -6398.389} C_VEL
LIN {X 0,Y 490.746,Z 411.099,A -85,B 0,C 180,E1 -6398.828,E2 -6398.828} C_VEL
LIN {X 0,Y 490.808,Z 420.737,A -85,B 0,C 180,E1 -6399.217,E2 -6399.217} C_VEL
LIN {X 0,Y 490.393,Z 432.009,A -85,B 0,C 180,E1 -6399.797,E2 -6399.797} C_VEL
LIN {X 0,Y 490.031,Z 443.096,A -85,B 0,C 180,E1 -6400.535,E2 -6400.535} C_VEL
LIN {X 0,Y 489.619,Z 453.29,A -85,B 0,C 180,E1 -6401.381,E2 -6401.381} C_VEL
LIN {X 0,Y 489.207,Z 463.525,A -85,B 0,C 180,E1 -6402.442,E2 -6402.442} C_VEL
LIN {X 0,Y 488.85,Z 471.887,A -85,B 0,C 180,E1 -6403.508,E2 -6403.508} C_VEL
LIN {X 0,Y 488.565,Z 480.062,A -85,B 0,C 180,E1 -6404.791,E2 -6404.791} C_VEL
LIN {X 0,Y 488.375,Z 485.591,A -85,B 0,C 180,E1 -6405.866,E2 -6405.866} C_VEL
LIN {X 0,Y 488.202,Z 490.995,A -85,B 0,C 180,E1 -6407.162,E2 -6407.162} C_VEL
LIN {X 0,Y 488.05,Z 495.173,A -85,B 0,C 180,E1 -6408.468,E2 -6408.468} C_VEL
LIN {X 0,Y 487.967,Z 497.307,A -85,B 0,C 180,E1 -6409.343,E2 -6409.343} C_VEL
LIN {X 0,Y 487.892,Z 499.515,A -85,B 0,C 180,E1 -6410.558,E2 -6410.558} C_VEL
LIN {X 0,Y 487.867,Z 500.978,A -85,B 0,C 180,E1 -6411.994,E2 -6411.994} C_VEL
LIN {X 0,Y 487.885,Z 501.3,A -85,B 0,C 180,E1 -6412.886,E2 -6412.886} C_VEL
LIN {X 0,Y 487.884,Z 501.166,A -85,B 0,C 180,E1 -6413.785,E2 -6413.785} C_VEL
LIN {X 0,Y 487.867,Z 500.4,A -85,B 0,C 180,E1 -6414.831,E2 -6414.831} C_VEL
LIN {X 0,Y 487.893,Z 499.451,A -85,B 0,C 180,E1 -6415.601,E2 -6415.601} C_VEL
LIN {X 0,Y 487.982,Z 497.33,A -85,B 0,C 180,E1 -6416.755,E2 -6416.755} C_VEL
LIN {X 0,Y 488.091,Z 494.415,A -85,B 0,C 180,E1 -6417.9,E2 -6417.9} C_VEL
LIN {X 0,Y 488.242,Z 489.642,A -85,B 0,C 180,E1 -6419.3,E2 -6419.3} C_VEL
LIN {X 0,Y 488.438,Z 483.554,A -85,B 0,C 180,E1 -6420.667,E2 -6420.667} C_VEL
LIN {X 0,Y 488.767,Z 476.14,A -85,B 0,C 180,E1 -6421.966,E2 -6421.966} C_VEL
LIN {X 0,Y 489.022,Z 468.171,A -85,B 0,C 180,E1 -6423.098,E2 -6423.098} C_VEL
LIN {X 0,Y 489.48,Z 458.861,A -85,B 0,C 180,E1 -6424.175,E2 -6424.175} C_VEL
LIN {X 0,Y 489.857,Z 448.568,A -85,B 0,C 180,E1 -6425.137,E2 -6425.137} C_VEL
LIN {X 0,Y 490.286,Z 437.022,A -85,B 0,C 180,E1 -6425.992,E2 -6425.992} C_VEL
LIN {X 0,Y 490.646,Z 425.407,A -85,B 0,C 180,E1 -6426.665,E2 -6426.665} C_VEL
LIN {X 0,Y 490.924,Z 412.527,A -85,B 0,C 180,E1 -6427.214,E2 -6427.214} C_VEL
LIN {X 0,Y 489.276,Z 404.133,A -85,B 0,C 180,E1 -6427.534,E2 -6427.534} C_VEL
LIN {X 0,Y 488.013,Z 398.893,A -85,B 0,C 180,E1 -6427.718,E2 -6427.718} C_VEL
LIN {X 0,Y 488.034,Z 396.007,A -85,B 0,C 180,E1 -6430.39,E2 -6430.39} C_VEL
LIN {X 0,Y 488.105,Z 393.456,A -85,B 0,C 180,E1 -6432.75,E2 -6432.75} C_VEL
LIN {X 0,Y 488.157,Z 389.981,A -85,B 0,C 180,E1 -6436.039,E2 -6436.039} C_VEL
LIN {X 0,Y 488.2,Z 387.311,A -85,B 0,C 180,E1 -6438.532,E2 -6438.532} C_VEL
LIN {X 0,Y 488.247,Z 383.919,A -85,B 0,C 180,E1 -6441.76,E2 -6441.76} C_VEL
LIN {X 0,Y 488.357,Z 380.361,A -85,B 0,C 180,E1 -6445.11,E2 -6445.11} C_VEL
LIN {X 0,Y 488.353,Z 379.659,A -85,B 0,C 180,E1 -6445.857,E2 -6445.857} C_VEL
LIN {X 0,Y 488.638,Z 379.624,A -85,B 0,C 180,E1 -6448.053,E2 -6448.053} C_VEL
LIN {X 0,Y 488.716,Z 379.611,A -85,B 0,C 180,E1 -6450.729,E2 -6450.729} C_VEL
LIN {X 0,Y 488.749,Z 379.607,A -85,B 0,C 180,E1 -6453.528,E2 -6453.528} C_VEL
LIN {X 0,Y 488.693,Z 379.615,A -85,B 0,C 180,E1 -6456.255,E2 -6456.255} C_VEL
LIN {X 0,Y 488.728,Z 379.61,A -85,B 0,C 180,E1 -6459.174,E2 -6459.174} C_VEL
LIN {X 0,Y 488.739,Z 379.608,A -85,B 0,C 180,E1 -6461.627,E2 -6461.627} C_VEL
LIN {X 0,Y 488.742,Z 379.606,A -85,B 0,C 180,E1 -6464.999,E2 -6464.999} C_VEL
LIN {X 0,Y 488.81,Z 379.599,A -85,B 0,C 180,E1 -6468.388,E2 -6468.388} C_VEL
LIN {X 0,Y 488.798,Z 379.599,A -85,B 0,C 180,E1 -6471.733,E2 -6471.733} C_VEL
LIN {X 0,Y 488.855,Z 379.593,A -85,B 0,C 180,E1 -6474.224,E2 -6474.224} C_VEL
LIN {X 0,Y 488.945,Z 379.58,A -85,B 0,C 180,E1 -6477.529,E2 -6477.529} C_VEL
LIN {X 0,Y 488.947,Z 379.58,A -85,B 0,C 180,E1 -6480,E2 -6480} C_VEL
LIN {X 0,Y 488.949,Z 379.58,A -85,B 0,C 180,E1 -6482.471,E2 -6482.471} C_VEL
LIN {X 0,Y 488.836,Z 379.594,A -85,B 0,C 180,E1 -6485.776,E2 -6485.776} C_VEL
LIN {X 0,Y 488.797,Z 379.599,A -85,B 0,C 180,E1 -6488.267,E2 -6488.267} C_VEL
LIN {X 0,Y 488.81,Z 379.6,A -85,B 0,C 180,E1 -6491.612,E2 -6491.612} C_VEL
LIN {X 0,Y 488.741,Z 379.606,A -85,B 0,C 180,E1 -6495.001,E2 -6495.001} C_VEL
LIN {X 0,Y 488.735,Z 379.609,A -85,B 0,C 180,E1 -6498.443,E2 -6498.443} C_VEL
LIN {X 0,Y 488.724,Z 379.612,A -85,B 0,C 180,E1 -6501.07,E2 -6501.07} C_VEL
LIN {X 0,Y 488.696,Z 379.616,A -85,B 0,C 180,E1 -6503.745,E2 -6503.745} C_VEL
LIN {X 0,Y 488.781,Z 379.603,A -85,B 0,C 180,E1 -6506.947,E2 -6506.947} C_VEL
LIN {X 0,Y 488.693,Z 379.616,A -85,B 0,C 180,E1 -6510.364,E2 -6510.364} C_VEL
LIN {X 0,Y 488.719,Z 379.61,A -85,B 0,C 180,E1 -6513.486,E2 -6513.486} C_VEL
LIN {X 0,Y 488.675,Z 379.615,A -85,B 0,C 180,E1 -6516.358,E2 -6516.358} C_VEL
LIN {X 0,Y 488.728,Z 379.609,A -85,B 0,C 180,E1 -6519.252,E2 -6519.252} C_VEL
LIN {X 0,Y 488.719,Z 379.614,A -85,B 0,C 180,E1 -6522.523,E2 -6522.523} C_VEL
LIN {X 0,Y 488.7,Z 379.618,A -85,B 0,C 180,E1 -6525.201,E2 -6525.201} C_VEL
LIN {X 0,Y 488.72,Z 379.613,A -85,B 0,C 180,E1 -6527.481,E2 -6527.481} C_VEL
LIN {X 0,Y 488.755,Z 379.645,A -85,B 0,C 180,E1 -6530.086,E2 -6530.086} C_VEL
LIN {X 0,Y 490.135,Z 387.423,A -85,B 0,C 180,E1 -6533.416,E2 -6533.416} C_VEL
LIN {X 0,Y 490.243,Z 391.488,A -85,B 0,C 180,E1 -6535.013,E2 -6535.013} C_VEL
LIN {X 0,Y 489.884,Z 399.369,A -85,B 0,C 180,E1 -6537.942,E2 -6537.942} C_VEL
LIN {X 0,Y 489.519,Z 408.445,A -85,B 0,C 180,E1 -6541.137,E2 -6541.137} C_VEL
LIN {X 0,Y 489.182,Z 418.128,A -85,B 0,C 180,E1 -6544.471,E2 -6544.471} C_VEL
LIN {X 0,Y 488.931,Z 427.86,A -85,B 0,C 180,E1 -6547.612,E2 -6547.612} C_VEL
LIN {X 0,Y 488.723,Z 437.47,A -85,B 0,C 180,E1 -6550.688,E2 -6550.688} C_VEL
LIN {X 0,Y 488.48,Z 446.737,A -85,B 0,C 180,E1 -6553.709,E2 -6553.709} C_VEL
LIN {X 0,Y 488.377,Z 451.651,A -85,B 0,C 180,E1 -6555.273,E2 -6555.273} C_VEL
LIN {X 0,Y 490.662,Z 465.16,A -85,B 0,C 180,E1 -6555.671,E2 -6555.671} C_VEL
LIN {X 0,Y 490.782,Z 470.556,A -85,B 0,C 180,E1 -6555.859,E2 -6555.859} C_VEL
LIN {X 0,Y 490.411,Z 483.54,A -85,B 0,C 180,E1 -6556.43,E2 -6556.43} C_VEL
LIN {X 0,Y 489.985,Z 495.432,A -85,B 0,C 180,E1 -6557.131,E2 -6557.131} C_VEL
LIN {X 0,Y 489.641,Z 506.765,A -85,B 0,C 180,E1 -6557.989,E2 -6557.989} C_VEL
LIN {X 0,Y 489.172,Z 517.615,A -85,B 0,C 180,E1 -6559.028,E2 -6559.028} C_VEL
LIN {X 0,Y 488.845,Z 526.427,A -85,B 0,C 180,E1 -6560.067,E2 -6560.067} C_VEL
LIN {X 0,Y 488.507,Z 535.014,A -85,B 0,C 180,E1 -6561.313,E2 -6561.313} C_VEL
LIN {X 0,Y 488.205,Z 541.877,A -85,B 0,C 180,E1 -6562.558,E2 -6562.558} C_VEL
LIN {X 0,Y 488.095,Z 547.069,A -85,B 0,C 180,E1 -6563.724,E2 -6563.724} C_VEL
LIN {X 0,Y 487.971,Z 551.682,A -85,B 0,C 180,E1 -6565.044,E2 -6565.044} C_VEL
LIN {X 0,Y 487.947,Z 553.962,A -85,B 0,C 180,E1 -6565.872,E2 -6565.872} C_VEL
LIN {X 0,Y 487.966,Z 555.81,A -85,B 0,C 180,E1 -6566.699,E2 -6566.699} C_VEL
LIN {X 0,Y 487.889,Z 558.184,A -85,B 0,C 180,E1 -6568.351,E2 -6568.351} C_VEL
LIN {X 0,Y 487.819,Z 559,A -85,B 0,C 180,E1 -6570.002,E2 -6570.002} C_VEL
LIN {X 0,Y 487.889,Z 558.183,A -85,B 0,C 180,E1 -6571.652,E2 -6571.652} C_VEL
LIN {X 0,Y 487.967,Z 555.807,A -85,B 0,C 180,E1 -6573.304,E2 -6573.304} C_VEL
LIN {X 0,Y 487.938,Z 552.891,A -85,B 0,C 180,E1 -6574.545,E2 -6574.545} C_VEL
LIN {X 0,Y 488.106,Z 548.943,A -85,B 0,C 180,E1 -6575.786,E2 -6575.786} C_VEL
LIN {X 0,Y 488.192,Z 542.869,A -85,B 0,C 180,E1 -6577.238,E2 -6577.238} C_VEL
LIN {X 0,Y 488.455,Z 536.227,A -85,B 0,C 180,E1 -6578.482,E2 -6578.482} C_VEL
LIN {X 0,Y 488.765,Z 527.982,A -85,B 0,C 180,E1 -6579.728,E2 -6579.728} C_VEL
LIN {X 0,Y 489.097,Z 519.527,A -85,B 0,C 180,E1 -6580.768,E2 -6580.768} C_VEL
LIN {X 0,Y 489.55,Z 509.077,A -85,B 0,C 180,E1 -6581.806,E2 -6581.806} C_VEL
LIN {X 0,Y 489.896,Z 497.868,A -85,B 0,C 180,E1 -6582.702,E2 -6582.702} C_VEL
LIN {X 0,Y 490.266,Z 487.383,A -85,B 0,C 180,E1 -6583.366,E2 -6583.366} C_VEL
LIN {X 0,Y 490.685,Z 475.731,A -85,B 0,C 180,E1 -6583.935,E2 -6583.935} C_VEL
LIN {X 0,Y 490.694,Z 465.477,A -85,B 0,C 180,E1 -6584.318,E2 -6584.318} C_VEL
LIN {X 0,Y 488.499,Z 452.508,A -85,B 0,C 180,E1 -6584.708,E2 -6584.708} C_VEL
LIN {X 0,Y 488.387,Z 451.526,A -85,B 0,C 180,E1 -6584.747,E2 -6584.747} C_VEL
LIN {X 0,Y 488.625,Z 441.609,A -85,B 0,C 180,E1 -6587.957,E2 -6587.957} C_VEL
LIN {X 0,Y 488.863,Z 432.03,A -85,B 0,C 180,E1 -6591.065,E2 -6591.065} C_VEL
LIN {X 0,Y 489.076,Z 422.36,A -85,B 0,C 180,E1 -6594.177,E2 -6594.177} C_VEL
LIN {X 0,Y 489.299,Z 415.555,A -85,B 0,C 180,E1 -6596.441,E2 -6596.441} C_VEL
LIN {X 0,Y 489.61,Z 406.292,A -85,B 0,C 180,E1 -6599.686,E2 -6599.686} C_VEL
LIN {X 0,Y 490.054,Z 396.984,A -85,B 0,C 180,E1 -6603.024,E2 -6603.024} C_VEL
LIN {X 0,Y 490.346,Z 390.194,A -85,B 0,C 180,E1 -6605.555,E2 -6605.555} C_VEL
LIN {X 0,Y 489.954,Z 386.459,A -85,B 0,C 180,E1 -6607.047,E2 -6607.047} C_VEL
LIN {X 0,Y 488.725,Z 379.611,A -85,B 0,C 180,E1 -6609.988,E2 -6609.988} C_VEL
LIN {X 0,Y 488.691,Z 379.614,A -85,B 0,C 180,E1 -6612.824,E2 -6612.824} C_VEL
LIN {X 0,Y 488.7,Z 379.613,A -85,B 0,C 180,E1 -6615.977,E2 -6615.977} C_VEL
LIN {X 0,Y 488.713,Z 379.612,A -85,B 0,C 180,E1 -6618.585,E2 -6618.585} C_VEL
LIN {X 0,Y 488.709,Z 379.612,A -85,B 0,C 180,E1 -6620.948,E2 -6620.948} C_VEL
LIN {X 0,Y 488.682,Z 379.614,A -85,B 0,C 180,E1 -6623.868,E2 -6623.868} C_VEL
LIN {X 0,Y 488.74,Z 379.609,A -85,B 0,C 180,E1 -6626.877,E2 -6626.877} C_VEL
LIN {X 0,Y 488.729,Z 379.607,A -85,B 0,C 180,E1 -6629.781,E2 -6629.781} C_VEL
LIN {X 0,Y 488.797,Z 379.601,A -85,B 0,C 180,E1 -6633.057,E2 -6633.057} C_VEL
LIN {X 0,Y 488.694,Z 379.614,A -85,B 0,C 180,E1 -6636.254,E2 -6636.254} C_VEL
LIN {X 0,Y 488.751,Z 379.606,A -85,B 0,C 180,E1 -6639.176,E2 -6639.176} C_VEL
LIN {X 0,Y 488.739,Z 379.609,A -85,B 0,C 180,E1 -6642.423,E2 -6642.423} C_VEL
LIN {X 0,Y 488.767,Z 379.603,A -85,B 0,C 180,E1 -6645,E2 -6645} C_VEL
LIN {X 0,Y 488.81,Z 379.599,A -85,B 0,C 180,E1 -6648.388,E2 -6648.388} C_VEL
LIN {X 0,Y 488.822,Z 379.597,A -85,B 0,C 180,E1 -6651.734,E2 -6651.734} C_VEL
LIN {X 0,Y 488.853,Z 379.594,A -85,B 0,C 180,E1 -6654.224,E2 -6654.224} C_VEL
LIN {X 0,Y 488.964,Z 379.579,A -85,B 0,C 180,E1 -6657.529,E2 -6657.529} C_VEL
LIN {X 0,Y 488.937,Z 379.582,A -85,B 0,C 180,E1 -6660.824,E2 -6660.824} C_VEL
LIN {X 0,Y 488.964,Z 379.579,A -85,B 0,C 180,E1 -6662.471,E2 -6662.471} C_VEL
LIN {X 0,Y 488.852,Z 379.594,A -85,B 0,C 180,E1 -6665.776,E2 -6665.776} C_VEL
LIN {X 0,Y 488.822,Z 379.598,A -85,B 0,C 180,E1 -6668.266,E2 -6668.266} C_VEL
LIN {X 0,Y 488.81,Z 379.6,A -85,B 0,C 180,E1 -6671.612,E2 -6671.612} C_VEL
LIN {X 0,Y 488.766,Z 379.603,A -85,B 0,C 180,E1 -6675,E2 -6675} C_VEL
LIN {X 0,Y 488.76,Z 379.605,A -85,B 0,C 180,E1 -6678.442,E2 -6678.442} C_VEL
LIN {X 0,Y 488.711,Z 379.611,A -85,B 0,C 180,E1 -6681.071,E2 -6681.071} C_VEL
LIN {X 0,Y 488.694,Z 379.615,A -85,B 0,C 180,E1 -6683.745,E2 -6683.745} C_VEL
LIN {X 0,Y 488.797,Z 379.6,A -85,B 0,C 180,E1 -6686.943,E2 -6686.943} C_VEL
LIN {X 0,Y 488.714,Z 379.609,A -85,B 0,C 180,E1 -6690.362,E2 -6690.362} C_VEL
LIN {X 0,Y 488.739,Z 379.608,A -85,B 0,C 180,E1 -6693.484,E2 -6693.484} C_VEL
LIN {X 0,Y 488.686,Z 379.613,A -85,B 0,C 180,E1 -6696.354,E2 -6696.354} C_VEL
LIN {X 0,Y 488.705,Z 379.613,A -85,B 0,C 180,E1 -6699.254,E2 -6699.254} C_VEL
LIN {X 0,Y 488.711,Z 379.611,A -85,B 0,C 180,E1 -6701.599,E2 -6701.599} C_VEL
LIN {X 0,Y 488.706,Z 379.613,A -85,B 0,C 180,E1 -6704.802,E2 -6704.802} C_VEL
LIN {X 0,Y 488.697,Z 379.614,A -85,B 0,C 180,E1 -6707.474,E2 -6707.474} C_VEL
LIN {X 0,Y 488.738,Z 379.608,A -85,B 0,C 180,E1 -6709.676,E2 -6709.676} C_VEL
LIN {X 0,Y 488.684,Z 379.615,A -85,B 0,C 180,E1 -6712.84,E2 -6712.84} C_VEL
LIN {X 0,Y 488.736,Z 379.607,A -85,B 0,C 180,E1 -6715.886,E2 -6715.886} C_VEL
LIN {X 0,Y 488.696,Z 379.613,A -85,B 0,C 180,E1 -6718.819,E2 -6718.819} C_VEL
LIN {X 0,Y 488.749,Z 379.605,A -85,B 0,C 180,E1 -6721.67,E2 -6721.67} C_VEL
LIN {X 0,Y 488.748,Z 379.606,A -85,B 0,C 180,E1 -6724.346,E2 -6724.346} C_VEL
LIN {X 0,Y 488.103,Z 379.691,A -85,B 0,C 180,E1 -6725.034,E2 -6725.034} C_VEL
LIN {X 0,Y 485.234,Z 380.048,A -85,B 0,C 180,E1 -6726.15,E2 -6726.15} C_VEL
LIN {X 0,Y 482.787,Z 380.349,A -85,B 0,C 180,E1 -6727.05,E2 -6727.05} C_VEL
LIN {X 0,Y 481.729,Z 380.479,A -85,B 0,C 180,E1 -6727.745,E2 -6727.745} C_VEL
LIN {X 0,Y 481.641,Z 380.489,A -85,B 0,C 180,E1 -6727.981,E2 -6727.981} C_VEL
LIN {X 0,Y 481.71,Z 380.483,A -85,B 0,C 180,E1 -6730.392,E2 -6730.392} C_VEL
LIN {X 0,Y 481.692,Z 380.485,A -85,B 0,C 180,E1 -6733.033,E2 -6733.033} C_VEL
LIN {X 0,Y 481.691,Z 380.484,A -85,B 0,C 180,E1 -6735.637,E2 -6735.637} C_VEL
LIN {X 0,Y 481.68,Z 380.488,A -85,B 0,C 180,E1 -6738.212,E2 -6738.212} C_VEL
LIN {X 0,Y 481.346,Z 380.531,A -85,B 0,C 180,E1 -6740.756,E2 -6740.756} C_VEL
LIN {X 0,Y 481.316,Z 382.779,A -85,B 0,C 180,E1 -6743.174,E2 -6743.174} C_VEL
LIN {X 0,Y 481.341,Z 385.571,A -85,B 0,C 180,E1 -6745.812,E2 -6745.812} C_VEL
LIN {X 0,Y 481.074,Z 390.078,A -85,B 0,C 180,E1 -6749.998,E2 -6749.998} C_VEL
LIN {X 0,Y 481.102,Z 393.679,A -85,B 0,C 180,E1 -6753.348,E2 -6753.348} C_VEL
LIN {X 0,Y 481.07,Z 397.374,A -85,B 0,C 180,E1 -6756.71,E2 -6756.71} C_VEL
LIN {X 0,Y 481.013,Z 398.972,A -85,B 0,C 180,E1 -6758.162,E2 -6758.162} C_VEL
LIN {X 0,Y 483.957,Z 412.679,A -85,B 0,C 180,E1 -6758.667,E2 -6758.667} C_VEL
LIN {X 0,Y 483.8,Z 424.904,A -85,B 0,C 180,E1 -6759.193,E2 -6759.193} C_VEL
LIN {X 0,Y 483.379,Z 436.131,A -85,B 0,C 180,E1 -6759.835,E2 -6759.835} C_VEL
LIN {X 0,Y 482.97,Z 447.741,A -85,B 0,C 180,E1 -6760.69,E2 -6760.69} C_VEL
LIN {X 0,Y 482.527,Z 458.221,A -85,B 0,C 180,E1 -6761.657,E2 -6761.657} C_VEL
LIN {X 0,Y 482.026,Z 468.456,A -85,B 0,C 180,E1 -6762.845,E2 -6762.845} C_VEL
LIN {X 0,Y 481.682,Z 477.405,A -85,B 0,C 180,E1 -6764.144,E2 -6764.144} C_VEL
LIN {X 0,Y 481.399,Z 484.864,A -85,B 0,C 180,E1 -6765.519,E2 -6765.519} C_VEL
LIN {X 0,Y 481.151,Z 491.07,A -85,B 0,C 180,E1 -6766.984,E2 -6766.984} C_VEL
LIN {X 0,Y 481.008,Z 495.16,A -85,B 0,C 180,E1 -6768.247,E2 -6768.247} C_VEL
LIN {X 0,Y 480.857,Z 498.48,A -85,B 0,C 180,E1 -6769.641,E2 -6769.641} C_VEL
LIN {X 0,Y 480.818,Z 500.176,A -85,B 0,C 180,E1 -6770.695,E2 -6770.695} C_VEL
LIN {X 0,Y 480.781,Z 501.613,A -85,B 0,C 180,E1 -6772.335,E2 -6772.335} C_VEL
LIN {X 0,Y 480.802,Z 501.728,A -85,B 0,C 180,E1 -6773.243,E2 -6773.243} C_VEL
LIN {X 0,Y 480.78,Z 501.398,A -85,B 0,C 180,E1 -6774.159,E2 -6774.159} C_VEL
LIN {X 0,Y 480.79,Z 500.618,A -85,B 0,C 180,E1 -6775.079,E2 -6775.079} C_VEL
LIN {X 0,Y 480.837,Z 499.299,A -85,B 0,C 180,E1 -6776.005,E2 -6776.005} C_VEL
LIN {X 0,Y 480.986,Z 496.385,A -85,B 0,C 180,E1 -6777.401,E2 -6777.401} C_VEL
LIN {X 0,Y 481.124,Z 492.186,A -85,B 0,C 180,E1 -6778.817,E2 -6778.817} C_VEL
LIN {X 0,Y 481.309,Z 486.97,A -85,B 0,C 180,E1 -6780.145,E2 -6780.145} C_VEL
LIN {X 0,Y 481.593,Z 480.456,A -85,B 0,C 180,E1 -6781.444,E2 -6781.444} C_VEL
LIN {X 0,Y 481.897,Z 472.908,A -85,B 0,C 180,E1 -6782.654,E2 -6782.654} C_VEL
LIN {X 0,Y 482.315,Z 463.756,A -85,B 0,C 180,E1 -6783.843,E2 -6783.843} C_VEL
LIN {X 0,Y 482.691,Z 454.189,A -85,B 0,C 180,E1 -6784.851,E2 -6784.851} C_VEL
LIN {X 0,Y 483.19,Z 442.443,A -85,B 0,C 180,E1 -6785.831,E2 -6785.831} C_VEL
LIN {X 0,Y 483.591,Z 431.208,A -85,B 0,C 180,E1 -6786.57,E2 -6786.57} C_VEL
LIN {X 0,Y 483.961,Z 418.845,A -85,B 0,C 180,E1 -6787.188,E2 -6787.188} C_VEL
LIN {X 0,Y 483.861,Z 411.642,A -85,B 0,C 180,E1 -6787.473,E2 -6787.473} C_VEL
LIN {X 0,Y 480.97,Z 399.324,A -85,B 0,C 180,E1 -6787.945,E2 -6787.945} C_VEL
LIN {X 0,Y 480.985,Z 395.913,A -85,B 0,C 180,E1 -6791.108,E2 -6791.108} C_VEL
LIN {X 0,Y 481.066,Z 392.531,A -85,B 0,C 180,E1 -6794.287,E2 -6794.287} C_VEL
LIN {X 0,Y 481.099,Z 389.759,A -85,B 0,C 180,E1 -6796.917,E2 -6796.917} C_VEL
LIN {X 0,Y 481.142,Z 386.525,A -85,B 0,C 180,E1 -6800.006,E2 -6800.006} C_VEL
LIN {X 0,Y 481.241,Z 382.932,A -85,B 0,C 180,E1 -6803.434,E2 -6803.434} C_VEL
LIN {X 0,Y 481.293,Z 380.98,A -85,B 0,C 180,E1 -6805.285,E2 -6805.285} C_VEL
LIN {X 0,Y 481.392,Z 380.526,A -85,B 0,C 180,E1 -6806.317,E2 -6806.317} C_VEL
LIN {X 0,Y 481.588,Z 380.502,A -85,B 0,C 180,E1 -6808.307,E2 -6808.307} C_VEL
LIN {X 0,Y 481.689,Z 380.486,A -85,B 0,C 180,E1 -6811.218,E2 -6811.218} C_VEL
LIN {X 0,Y 481.689,Z 380.486,A -85,B 0,C 180,E1 -6814.042,E2 -6814.042} C_VEL
LIN {X 0,Y 481.673,Z 380.488,A -85,B 0,C 180,E1 -6816.806,E2 -6816.806} C_VEL
LIN {X 0,Y 481.679,Z 380.485,A -85,B 0,C 180,E1 -6819.502,E2 -6819.502} C_VEL
LIN {X 0,Y 481.687,Z 380.485,A -85,B 0,C 180,E1 -6822.158,E2 -6822.158} C_VEL
LIN {X 0,Y 481.722,Z 380.482,A -85,B 0,C 180,E1 -6824.775,E2 -6824.775} C_VEL
LIN {X 0,Y 481.775,Z 380.474,A -85,B 0,C 180,E1 -6828.216,E2 -6828.216} C_VEL
LIN {X 0,Y 481.744,Z 380.478,A -85,B 0,C 180,E1 -6831.611,E2 -6831.611} C_VEL
LIN {X 0,Y 481.813,Z 380.471,A -85,B 0,C 180,E1 -6834.14,E2 -6834.14} C_VEL
LIN {X 0,Y 481.911,Z 380.456,A -85,B 0,C 180,E1 -6837.493,E2 -6837.493} C_VEL
LIN {X 0,Y 481.918,Z 380.455,A -85,B 0,C 180,E1 -6840,E2 -6840} C_VEL
LIN {X 0,Y 481.916,Z 380.456,A -85,B 0,C 180,E1 -6842.508,E2 -6842.508} C_VEL
LIN {X 0,Y 481.797,Z 380.471,A -85,B 0,C 180,E1 -6845.861,E2 -6845.861} C_VEL
LIN {X 0,Y 481.743,Z 380.478,A -85,B 0,C 180,E1 -6848.389,E2 -6848.389} C_VEL
LIN {X 0,Y 481.775,Z 380.475,A -85,B 0,C 180,E1 -6851.784,E2 -6851.784} C_VEL
LIN {X 0,Y 481.722,Z 380.481,A -85,B 0,C 180,E1 -6855.225,E2 -6855.225} C_VEL
LIN {X 0,Y 481.693,Z 380.484,A -85,B 0,C 180,E1 -6858.723,E2 -6858.723} C_VEL
LIN {X 0,Y 481.659,Z 380.489,A -85,B 0,C 180,E1 -6861.394,E2 -6861.394} C_VEL
LIN {X 0,Y 481.674,Z 380.488,A -85,B 0,C 180,E1 -6864.113,E2 -6864.113} C_VEL
LIN {X 0,Y 481.734,Z 380.48,A -85,B 0,C 180,E1 -6867.142,E2 -6867.142} C_VEL
LIN {X 0,Y 481.661,Z 380.489,A -85,B 0,C 180,E1 -6869.742,E2 -6869.742} C_VEL
LIN {X 0,Y 481.657,Z 380.489,A -85,B 0,C 180,E1 -6872.676,E2 -6872.676} C_VEL
LIN {X 0,Y 481.628,Z 380.494,A -85,B 0,C 180,E1 -6875.71,E2 -6875.71} C_VEL
LIN {X 0,Y 481.7,Z 380.484,A -85,B 0,C 180,E1 -6879.356,E2 -6879.356} C_VEL
LIN {X 0,Y 481.661,Z 380.491,A -85,B 0,C 180,E1 -6882.159,E2 -6882.159} C_VEL
LIN {X 0,Y 481.647,Z 380.496,A -85,B 0,C 180,E1 -6884.459,E2 -6884.459} C_VEL
LIN {X 0,Y 481.677,Z 380.493,A -85,B 0,C 180,E1 -6886.848,E2 -6886.848} C_VEL
LIN {X 0,Y 481.721,Z 380.563,A -85,B 0,C 180,E1 -6889.805,E2 -6889.805} C_VEL
LIN {X 0,Y 483.097,Z 388.156,A -85,B 0,C 180,E1 -6893.143,E2 -6893.143} C_VEL
LIN {X 0,Y 483.276,Z 392.724,A -85,B 0,C 180,E1 -6894.985,E2 -6894.985} C_VEL
LIN {X 0,Y 482.878,Z 400.74,A -85,B 0,C 180,E1 -6897.986,E2 -6897.986} C_VEL
LIN {X 0,Y 482.474,Z 409.863,A -85,B 0,C 180,E1 -6901.272,E2 -6901.272} C_VEL
LIN {X 0,Y 482.194,Z 417.878,A -85,B 0,C 180,E1 -6904.074,E2 -6904.074} C_VEL
LIN {X 0,Y 481.925,Z 426.115,A -85,B 0,C 180,E1 -6906.814,E2 -6906.814} C_VEL
LIN {X 0,Y 481.714,Z 435.824,A -85,B 0,C 180,E1 -6909.951,E2 -6909.951} C_VEL
LIN {X 0,Y 481.5,Z 444.083,A -85,B 0,C 180,E1 -6912.591,E2 -6912.591} C_VEL
LIN {X 0,Y 481.325,Z 451.583,A -85,B 0,C 180,E1 -6915.05,E2 -6915.05} C_VEL
LIN {X 0,Y 483.612,Z 465.16,A -85,B 0,C 180,E1 -6915.457,E2 -6915.457} C_VEL
LIN {X 0,Y 483.985,Z 469.796,A -85,B 0,C 180,E1 -6915.63,E2 -6915.63} C_VEL
LIN {X 0,Y 483.558,Z 482.546,A -85,B 0,C 180,E1 -6916.18,E2 -6916.18} C_VEL
LIN {X 0,Y 483.089,Z 494.706,A -85,B 0,C 180,E1 -6916.895,E2 -6916.895} C_VEL
LIN {X 0,Y 482.754,Z 505.508,A -85,B 0,C 180,E1 -6917.709,E2 -6917.709} C_VEL
LIN {X 0,Y 482.319,Z 515.663,A -85,B 0,C 180,E1 -6918.657,E2 -6918.657} C_VEL
LIN {X 0,Y 481.876,Z 524.8,A -85,B 0,C 180,E1 -6919.71,E2 -6919.71} C_VEL
LIN {X 0,Y 481.529,Z 533.699,A -85,B 0,C 180,E1 -6920.975,E2 -6920.975} C_VEL
LIN {X 0,Y 481.206,Z 540.857,A -85,B 0,C 180,E1 -6922.238,E2 -6922.238} C_VEL
LIN {X 0,Y 481.046,Z 546.364,A -85,B 0,C 180,E1 -6923.449,E2 -6923.449} C_VEL
LIN {X 0,Y 480.998,Z 550.379,A -85,B 0,C 180,E1 -6924.552,E2 -6924.552} C_VEL
LIN {X 0,Y 480.846,Z 553.962,A -85,B 0,C 180,E1 -6925.811,E2 -6925.811} C_VEL
LIN {X 0,Y 480.891,Z 555.81,A -85,B 0,C 180,E1 -6926.65,E2 -6926.65} C_VEL
LIN {X 0,Y 480.789,Z 558.184,A -85,B 0,C 180,E1 -6928.326,E2 -6928.326} C_VEL
LIN {X 0,Y 480.743,Z 559,A -85,B 0,C 180,E1 -6930.002,E2 -6930.002} C_VEL
LIN {X 0,Y 480.79,Z 558.182,A -85,B 0,C 180,E1 -6931.677,E2 -6931.677} C_VEL
LIN {X 0,Y 480.892,Z 555.807,A -85,B 0,C 180,E1 -6933.353,E2 -6933.353} C_VEL
LIN {X 0,Y 480.854,Z 552.891,A -85,B 0,C 180,E1 -6934.612,E2 -6934.612} C_VEL
LIN {X 0,Y 481.024,Z 548.943,A -85,B 0,C 180,E1 -6935.872,E2 -6935.872} C_VEL
LIN {X 0,Y 481.118,Z 542.868,A -85,B 0,C 180,E1 -6937.345,E2 -6937.345} C_VEL
LIN {X 0,Y 481.427,Z 536.227,A -85,B 0,C 180,E1 -6938.607,E2 -6938.607} C_VEL
LIN {X 0,Y 481.757,Z 527.982,A -85,B 0,C 180,E1 -6939.871,E2 -6939.871} C_VEL
LIN {X 0,Y 482.113,Z 519.527,A -85,B 0,C 180,E1 -6940.925,E2 -6940.925} C_VEL
LIN {X 0,Y 482.589,Z 509.076,A -85,B 0,C 180,E1 -6941.979,E2 -6941.979} C_VEL
LIN {X 0,Y 482.971,Z 497.859,A -85,B 0,C 180,E1 -6942.888,E2 -6942.888} C_VEL
LIN {X 0,Y 483.438,Z 485.461,A -85,B 0,C 180,E1 -6943.666,E2 -6943.666} C_VEL
LIN {X 0,Y 483.876,Z 473.131,A -85,B 0,C 180,E1 -6944.243,E2 -6944.243} C_VEL
LIN {X 0,Y 483.724,Z 465.882,A -85,B 0,C 180,E1 -6944.516,E2 -6944.516} C_VEL
LIN {X 0,Y 481.563,Z 453.072,A -85,B 0,C 180,E1 -6944.915,E2 -6944.915} C_VEL
LIN {X 0,Y 481.328,Z 451.526,A -85,B 0,C 180,E1 -6944.968,E2 -6944.968} C_VEL
LIN {X 0,Y 481.554,Z 442.709,A -85,B 0,C 180,E1 -6947.849,E2 -6947.849} C_VEL
LIN {X 0,Y 481.799,Z 432.916,A -85,B 0,C 180,E1 -6951.002,E2 -6951.002} C_VEL
LIN {X 0,Y 482.014,Z 423.435,A -85,B 0,C 180,E1 -6954.096,E2 -6954.096} C_VEL
LIN {X 0,Y 482.287,Z 415.346,A -85,B 0,C 180,E1 -6956.857,E2 -6956.857} C_VEL
LIN {X 0,Y 482.654,Z 406.078,A -85,B 0,C 180,E1 -6960.157,E2 -6960.157} C_VEL
LIN {X 0,Y 483.066,Z 398.097,A -85,B 0,C 180,E1 -6963.065,E2 -6963.065} C_VEL
LIN {X 0,Y 483.376,Z 391.568,A -85,B 0,C 180,E1 -6965.563,E2 -6965.563} C_VEL
LIN {X 0,Y 482.919,Z 387.462,A -85,B 0,C 180,E1 -6967.227,E2 -6967.227} C_VEL
LIN {X 0,Y 481.721,Z 380.483,A -85,B 0,C 180,E1 -6970.263,E2 -6970.263} C_VEL
LIN {X 0,Y 481.637,Z 380.493,A -85,B 0,C 180,E1 -6973.301,E2 -6973.301} C_VEL
LIN {X 0,Y 481.66,Z 380.491,A -85,B 0,C 180,E1 -6975.642,E2 -6975.642} C_VEL
LIN {X 0,Y 481.662,Z 380.49,A -85,B 0,C 180,E1 -6978.959,E2 -6978.959} C_VEL
LIN {X 0,Y 481.659,Z 380.489,A -85,B 0,C 180,E1 -6981.993,E2 -6981.993} C_VEL
LIN {X 0,Y 481.69,Z 380.485,A -85,B 0,C 180,E1 -6985.318,E2 -6985.318} C_VEL
LIN {X 0,Y 481.65,Z 380.491,A -85,B 0,C 180,E1 -6988.312,E2 -6988.312} C_VEL
LIN {X 0,Y 481.705,Z 380.483,A -85,B 0,C 180,E1 -6991.219,E2 -6991.219} C_VEL
LIN {X 0,Y 481.706,Z 380.483,A -85,B 0,C 180,E1 -6994.043,E2 -6994.043} C_VEL
LIN {X 0,Y 481.68,Z 380.487,A -85,B 0,C 180,E1 -6996.812,E2 -6996.812} C_VEL
LIN {X 0,Y 481.701,Z 380.483,A -85,B 0,C 180,E1 -6999.503,E2 -6999.503} C_VEL
LIN {X 0,Y 481.712,Z 380.483,A -85,B 0,C 180,E1 -7002.159,E2 -7002.159} C_VEL
LIN {X 0,Y 481.748,Z 380.478,A -85,B 0,C 180,E1 -7004.776,E2 -7004.776} C_VEL
LIN {X 0,Y 481.755,Z 380.478,A -85,B 0,C 180,E1 -7008.215,E2 -7008.215} C_VEL
LIN {X 0,Y 481.768,Z 380.474,A -85,B 0,C 180,E1 -7011.612,E2 -7011.612} C_VEL
LIN {X 0,Y 481.814,Z 380.471,A -85,B 0,C 180,E1 -7014.139,E2 -7014.139} C_VEL
LIN {X 0,Y 481.931,Z 380.455,A -85,B 0,C 180,E1 -7017.492,E2 -7017.492} C_VEL
LIN {X 0,Y 481.889,Z 380.46,A -85,B 0,C 180,E1 -7020.836,E2 -7020.836} C_VEL
LIN {X 0,Y 481.931,Z 380.455,A -85,B 0,C 180,E1 -7022.507,E2 -7022.507} C_VEL
LIN {X 0,Y 481.812,Z 380.471,A -85,B 0,C 180,E1 -7025.86,E2 -7025.86} C_VEL
LIN {X 0,Y 481.768,Z 380.476,A -85,B 0,C 180,E1 -7028.388,E2 -7028.388} C_VEL
LIN {X 0,Y 481.755,Z 380.478,A -85,B 0,C 180,E1 -7031.785,E2 -7031.785} C_VEL
LIN {X 0,Y 481.747,Z 380.478,A -85,B 0,C 180,E1 -7035.224,E2 -7035.224} C_VEL
LIN {X 0,Y 481.717,Z 380.481,A -85,B 0,C 180,E1 -7038.721,E2 -7038.721} C_VEL
LIN {X 0,Y 481.65,Z 380.491,A -85,B 0,C 180,E1 -7041.395,E2 -7041.395} C_VEL
LIN {X 0,Y 481.678,Z 380.486,A -85,B 0,C 180,E1 -7044.113,E2 -7044.113} C_VEL
LIN {X 0,Y 481.752,Z 380.479,A -85,B 0,C 180,E1 -7047.139,E2 -7047.139} C_VEL
LIN {X 0,Y 481.683,Z 380.487,A -85,B 0,C 180,E1 -7049.741,E2 -7049.741} C_VEL
LIN {X 0,Y 481.676,Z 380.486,A -85,B 0,C 180,E1 -7052.674,E2 -7052.674} C_VEL
LIN {X 0,Y 481.641,Z 380.492,A -85,B 0,C 180,E1 -7055.709,E2 -7055.709} C_VEL
LIN {X 0,Y 481.675,Z 380.487,A -85,B 0,C 180,E1 -7058.859,E2 -7058.859} C_VEL
LIN {X 0,Y 481.657,Z 380.488,A -85,B 0,C 180,E1 -7061.912,E2 -7061.912} C_VEL
LIN {X 0,Y 481.659,Z 380.488,A -85,B 0,C 180,E1 -7064.457,E2 -7064.457} C_VEL
LIN {X 0,Y 481.653,Z 380.489,A -85,B 0,C 180,E1 -7067.839,E2 -7067.839} C_VEL
LIN {X 0,Y 481.686,Z 380.486,A -85,B 0,C 180,E1 -7070.651,E2 -7070.651} C_VEL
LIN {X 0,Y 481.633,Z 380.493,A -85,B 0,C 180,E1 -7073.376,E2 -7073.376} C_VEL
LIN {X 0,Y 481.715,Z 380.482,A -85,B 0,C 180,E1 -7076.329,E2 -7076.329} C_VEL
LIN {X 0,Y 481.655,Z 380.489,A -85,B 0,C 180,E1 -7079.417,E2 -7079.417} C_VEL
LIN {X 0,Y 481.704,Z 380.483,A -85,B 0,C 180,E1 -7082.167,E2 -7082.167} C_VEL
LIN {X 0,Y 481.723,Z 380.482,A -85,B 0,C 180,E1 -7084.969,E2 -7084.969} C_VEL
LIN {X 0,Y 481.641,Z 380.489,A -85,B 0,C 180,E1 -7087.981,E2 -7087.981} C_VEL
LIN {X 0,Y 480.974,Z 380.576,A -85,B 0,C 180,E1 -7088.679,E2 -7088.679} C_VEL
LIN {X 0,Y 478.148,Z 380.926,A -85,B 0,C 180,E1 -7089.813,E2 -7089.813} C_VEL
LIN {X 0,Y 475.763,Z 381.225,A -85,B 0,C 180,E1 -7090.727,E2 -7090.727} C_VEL
LIN {X 0,Y 474.742,Z 381.35,A -85,B 0,C 180,E1 -7091.433,E2 -7091.433} C_VEL
LIN {X 0,Y 474.659,Z 381.36,A -85,B 0,C 180,E1 -7091.672,E2 -7091.672} C_VEL
LIN {X 0,Y 474.705,Z 381.357,A -85,B 0,C 180,E1 -7094.543,E2 -7094.543} C_VEL
LIN {X 0,Y 474.651,Z 381.363,A -85,B 0,C 180,E1 -7098.035,E2 -7098.035} C_VEL
LIN {X 0,Y 474.331,Z 381.405,A -85,B 0,C 180,E1 -7100.618,E2 -7100.618} C_VEL
LIN {X 0,Y 474.235,Z 381.758,A -85,B 0,C 180,E1 -7101.476,E2 -7101.476} C_VEL
LIN {X 0,Y 474.172,Z 384.412,A -85,B 0,C 180,E1 -7104.043,E2 -7104.043} C_VEL
LIN {X 0,Y 474.299,Z 386.23,A -85,B 0,C 180,E1 -7105.75,E2 -7105.75} C_VEL
LIN {X 0,Y 474.003,Z 390.75,A -85,B 0,C 180,E1 -7109.998,E2 -7109.998} C_VEL
LIN {X 0,Y 474.052,Z 394.445,A -85,B 0,C 180,E1 -7113.398,E2 -7113.398} C_VEL
LIN {X 0,Y 474.001,Z 398.101,A -85,B 0,C 180,E1 -7116.81,E2 -7116.81} C_VEL
LIN {X 0,Y 473.935,Z 399.354,A -85,B 0,C 180,E1 -7117.933,E2 -7117.933} C_VEL
LIN {X 0,Y 477.043,Z 413.489,A -85,B 0,C 180,E1 -7118.47,E2 -7118.47} C_VEL
LIN {X 0,Y 476.985,Z 423.835,A -85,B 0,C 180,E1 -7118.92,E2 -7118.92} C_VEL
LIN {X 0,Y 476.52,Z 435.139,A -85,B 0,C 180,E1 -7119.549,E2 -7119.549} C_VEL
LIN {X 0,Y 476.125,Z 445.749,A -85,B 0,C 180,E1 -7120.308,E2 -7120.308} C_VEL
LIN {X 0,Y 475.642,Z 456.64,A -85,B 0,C 180,E1 -7121.288,E2 -7121.288} C_VEL
LIN {X 0,Y 475.198,Z 466.343,A -85,B 0,C 180,E1 -7122.37,E2 -7122.37} C_VEL
LIN {X 0,Y 474.798,Z 474.466,A -85,B 0,C 180,E1 -7123.48,E2 -7123.48} C_VEL
LIN {X 0,Y 474.483,Z 482.255,A -85,B 0,C 180,E1 -7124.802,E2 -7124.802} C_VEL
LIN {X 0,Y 474.264,Z 487.642,A -85,B 0,C 180,E1 -7125.924,E2 -7125.924} C_VEL
LIN {X 0,Y 474.052,Z 492.719,A -85,B 0,C 180,E1 -7127.246,E2 -7127.246} C_VEL
LIN {X 0,Y 473.941,Z 496.12,A -85,B 0,C 180,E1 -7128.369,E2 -7128.369} C_VEL
LIN {X 0,Y 473.757,Z 499.532,A -85,B 0,C 180,E1 -7129.948,E2 -7129.948} C_VEL
LIN {X 0,Y 473.736,Z 500.861,A -85,B 0,C 180,E1 -7130.855,E2 -7130.855} C_VEL
LIN {X 0,Y 473.687,Z 501.734,A -85,B 0,C 180,E1 -7131.77,E2 -7131.77} C_VEL
LIN {X 0,Y 473.722,Z 502.186,A -85,B 0,C 180,E1 -7133.101,E2 -7133.101} C_VEL
LIN {X 0,Y 473.707,Z 501.583,A -85,B 0,C 180,E1 -7134.543,E2 -7134.543} C_VEL
LIN {X 0,Y 473.738,Z 500.577,A -85,B 0,C 180,E1 -7135.479,E2 -7135.479} C_VEL
LIN {X 0,Y 473.783,Z 499.109,A -85,B 0,C 180,E1 -7136.422,E2 -7136.422} C_VEL
LIN {X 0,Y 473.969,Z 495.867,A -85,B 0,C 180,E1 -7137.843,E2 -7137.843} C_VEL
LIN {X 0,Y 474.122,Z 491.274,A -85,B 0,C 180,E1 -7139.283,E2 -7139.283} C_VEL
LIN {X 0,Y 474.367,Z 485.051,A -85,B 0,C 180,E1 -7140.762,E2 -7140.762} C_VEL
LIN {X 0,Y 474.679,Z 478.693,A -85,B 0,C 180,E1 -7141.956,E2 -7141.956} C_VEL
LIN {X 0,Y 475.031,Z 470.623,A -85,B 0,C 180,E1 -7143.187,E2 -7143.187} C_VEL
LIN {X 0,Y 475.484,Z 461.62,A -85,B 0,C 180,E1 -7144.296,E2 -7144.296} C_VEL
LIN {X 0,Y 475.926,Z 451.028,A -85,B 0,C 180,E1 -7145.356,E2 -7145.356} C_VEL
LIN {X 0,Y 476.393,Z 440.985,A -85,B 0,C 180,E1 -7146.161,E2 -7146.161} C_VEL
LIN {X 0,Y 476.798,Z 429.077,A -85,B 0,C 180,E1 -7146.914,E2 -7146.914} C_VEL
LIN {X 0,Y 477.172,Z 415.957,A -85,B 0,C 180,E1 -7147.534,E2 -7147.534} C_VEL
LIN {X 0,Y 476.81,Z 411.933,A -85,B 0,C 180,E1 -7147.697,E2 -7147.697} C_VEL
LIN {X 0,Y 473.891,Z 399.776,A -85,B 0,C 180,E1 -7148.159,E2 -7148.159} C_VEL
LIN {X 0,Y 473.903,Z 396.889,A -85,B 0,C 180,E1 -7150.858,E2 -7150.858} C_VEL
LIN {X 0,Y 474.011,Z 394.194,A -85,B 0,C 180,E1 -7153.406,E2 -7153.406} C_VEL
LIN {X 0,Y 474.045,Z 390.843,A -85,B 0,C 180,E1 -7156.586,E2 -7156.586} C_VEL
LIN {X 0,Y 474.088,Z 388.021,A -85,B 0,C 180,E1 -7159.287,E2 -7159.287} C_VEL
LIN {X 0,Y 474.148,Z 384.611,A -85,B 0,C 180,E1 -7162.575,E2 -7162.575} C_VEL
LIN {X 0,Y 474.256,Z 381.415,A -85,B 0,C 180,E1 -7165.728,E2 -7165.728} C_VEL
LIN {X 0,Y 474.531,Z 381.382,A -85,B 0,C 180,E1 -7167.78,E2 -7167.78} C_VEL
LIN {X 0,Y 474.614,Z 381.368,A -85,B 0,C 180,E1 -7170.882,E2 -7170.882} C_VEL
LIN {X 0,Y 474.649,Z 381.364,A -85,B 0,C 180,E1 -7173.628,E2 -7173.628} C_VEL
LIN {X 0,Y 474.634,Z 381.366,A -85,B 0,C 180,E1 -7176.635,E2 -7176.635} C_VEL
LIN {X 0,Y 474.657,Z 381.362,A -85,B 0,C 180,E1 -7179.185,E2 -7179.185} C_VEL
LIN {X 0,Y 474.637,Z 381.364,A -85,B 0,C 180,E1 -7181.884,E2 -7181.884} C_VEL
LIN {X 0,Y 474.679,Z 381.359,A -85,B 0,C 180,E1 -7184.544,E2 -7184.544} C_VEL
LIN {X 0,Y 474.719,Z 381.352,A -85,B 0,C 180,E1 -7188.038,E2 -7188.038} C_VEL
LIN {X 0,Y 474.709,Z 381.355,A -85,B 0,C 180,E1 -7191.486,E2 -7191.486} C_VEL
LIN {X 0,Y 474.773,Z 381.348,A -85,B 0,C 180,E1 -7194.052,E2 -7194.052} C_VEL
LIN {X 0,Y 474.877,Z 381.332,A -85,B 0,C 180,E1 -7197.455,E2 -7197.455} C_VEL
LIN {X 0,Y 474.889,Z 381.331,A -85,B 0,C 180,E1 -7200,E2 -7200} C_VEL
LIN {X 0,Y 474.883,Z 381.332,A -85,B 0,C 180,E1 -7202.545,E2 -7202.545} C_VEL
LIN {X 0,Y 474.759,Z 381.349,A -85,B 0,C 180,E1 -7205.948,E2 -7205.948} C_VEL
LIN {X 0,Y 474.708,Z 381.354,A -85,B 0,C 180,E1 -7208.514,E2 -7208.514} C_VEL
LIN {X 0,Y 474.719,Z 381.353,A -85,B 0,C 180,E1 -7211.962,E2 -7211.962} C_VEL
LIN {X 0,Y 474.66,Z 381.362,A -85,B 0,C 180,E1 -7215.769,E2 -7215.769} C_VEL
LIN {X 0,Y 474.646,Z 381.361,A -85,B 0,C 180,E1 -7219.011,E2 -7219.011} C_VEL
LIN {X 0,Y 474.627,Z 381.365,A -85,B 0,C 180,E1 -7221.727,E2 -7221.727} C_VEL
LIN {X 0,Y 474.651,Z 381.362,A -85,B 0,C 180,E1 -7224.493,E2 -7224.493} C_VEL
LIN {X 0,Y 474.681,Z 381.359,A -85,B 0,C 180,E1 -7227.34,E2 -7227.34} C_VEL
LIN {X 0,Y 474.588,Z 381.371,A -85,B 0,C 180,E1 -7230.812,E2 -7230.812} C_VEL
LIN {X 0,Y 474.622,Z 381.365,A -85,B 0,C 180,E1 -7233.986,E2 -7233.986} C_VEL
LIN {X 0,Y 474.562,Z 381.373,A -85,B 0,C 180,E1 -7236.902,E2 -7236.902} C_VEL
LIN {X 0,Y 474.636,Z 381.365,A -85,B 0,C 180,E1 -7239.653,E2 -7239.653} C_VEL
LIN {X 0,Y 474.639,Z 381.369,A -85,B 0,C 180,E1 -7242.932,E2 -7242.932} C_VEL
LIN {X 0,Y 474.606,Z 381.373,A -85,B 0,C 180,E1 -7245.898,E2 -7245.898} C_VEL
LIN {X 0,Y 474.635,Z 381.367,A -85,B 0,C 180,E1 -7249.04,E2 -7249.04} C_VEL
LIN {X 0,Y 474.654,Z 381.385,A -85,B 0,C 180,E1 -7249.477,E2 -7249.477} C_VEL
LIN {X 0,Y 476.03,Z 388.876,A -85,B 0,C 180,E1 -7252.868,E2 -7252.868} C_VEL
LIN {X 0,Y 476.338,Z 392.215,A -85,B 0,C 180,E1 -7254.241,E2 -7254.241} C_VEL
LIN {X 0,Y 476.048,Z 398.993,A -85,B 0,C 180,E1 -7256.893,E2 -7256.893} C_VEL
LIN {X 0,Y 475.599,Z 406.937,A -85,B 0,C 180,E1 -7259.842,E2 -7259.842} C_VEL
LIN {X 0,Y 475.292,Z 414.959,A -85,B 0,C 180,E1 -7262.719,E2 -7262.719} C_VEL
LIN {X 0,Y 474.956,Z 424.366,A -85,B 0,C 180,E1 -7265.991,E2 -7265.991} C_VEL
LIN {X 0,Y 474.702,Z 434.092,A -85,B 0,C 180,E1 -7269.189,E2 -7269.189} C_VEL
LIN {X 0,Y 474.461,Z 443.746,A -85,B 0,C 180,E1 -7272.325,E2 -7272.325} C_VEL
LIN {X 0,Y 474.283,Z 451.562,A -85,B 0,C 180,E1 -7274.826,E2 -7274.826} C_VEL
LIN {X 0,Y 476.514,Z 464.591,A -85,B 0,C 180,E1 -7275.219,E2 -7275.219} C_VEL
LIN {X 0,Y 477.106,Z 469.796,A -85,B 0,C 180,E1 -7275.418,E2 -7275.418} C_VEL
LIN {X 0,Y 476.661,Z 482.545,A -85,B 0,C 180,E1 -7275.976,E2 -7275.976} C_VEL
LIN {X 0,Y 476.183,Z 494.705,A -85,B 0,C 180,E1 -7276.702,E2 -7276.702} C_VEL
LIN {X 0,Y 475.792,Z 505.556,A -85,B 0,C 180,E1 -7277.53,E2 -7277.53} C_VEL
LIN {X 0,Y 475.359,Z 515.663,A -85,B 0,C 180,E1 -7278.489,E2 -7278.489} C_VEL
LIN {X 0,Y 474.878,Z 524.8,A -85,B 0,C 180,E1 -7279.557,E2 -7279.557} C_VEL
LIN {X 0,Y 474.48,Z 533.699,A -85,B 0,C 180,E1 -7280.84,E2 -7280.84} C_VEL
LIN {X 0,Y 474.151,Z 540.857,A -85,B 0,C 180,E1 -7282.121,E2 -7282.121} C_VEL
LIN {X 0,Y 473.976,Z 546.726,A -85,B 0,C 180,E1 -7283.445,E2 -7283.445} C_VEL
LIN {X 0,Y 473.845,Z 551.682,A -85,B 0,C 180,E1 -7284.896,E2 -7284.896} C_VEL
LIN {X 0,Y 473.751,Z 553.962,A -85,B 0,C 180,E1 -7285.748,E2 -7285.748} C_VEL
LIN {X 0,Y 473.799,Z 555.81,A -85,B 0,C 180,E1 -7286.6,E2 -7286.6} C_VEL
LIN {X 0,Y 473.695,Z 558.183,A -85,B 0,C 180,E1 -7288.301,E2 -7288.301} C_VEL
LIN {X 0,Y 473.688,Z 558.786,A -85,B 0,C 180,E1 -7289.152,E2 -7289.152} C_VEL
LIN {X 0,Y 473.669,Z 559,A -85,B 0,C 180,E1 -7290.002,E2 -7290.002} C_VEL
LIN {X 0,Y 473.688,Z 558.785,A -85,B 0,C 180,E1 -7290.852,E2 -7290.852} C_VEL
LIN {X 0,Y 473.724,Z 557.194,A -85,B 0,C 180,E1 -7292.552,E2 -7292.552} C_VEL
LIN {X 0,Y 473.8,Z 555.807,A -85,B 0,C 180,E1 -7293.403,E2 -7293.403} C_VEL
LIN {X 0,Y 473.776,Z 552.891,A -85,B 0,C 180,E1 -7294.681,E2 -7294.681} C_VEL
LIN {X 0,Y 473.943,Z 548.943,A -85,B 0,C 180,E1 -7295.96,E2 -7295.96} C_VEL
LIN {X 0,Y 474.051,Z 542.868,A -85,B 0,C 180,E1 -7297.455,E2 -7297.455} C_VEL
LIN {X 0,Y 474.379,Z 536.227,A -85,B 0,C 180,E1 -7298.736,E2 -7298.736} C_VEL
LIN {X 0,Y 474.753,Z 527.982,A -85,B 0,C 180,E1 -7300.018,E2 -7300.018} C_VEL
LIN {X 0,Y 475.124,Z 519.527,A -85,B 0,C 180,E1 -7301.088,E2 -7301.088} C_VEL
LIN {X 0,Y 475.648,Z 509.097,A -85,B 0,C 180,E1 -7302.154,E2 -7302.154} C_VEL
LIN {X 0,Y 476.031,Z 498.022,A -85,B 0,C 180,E1 -7303.067,E2 -7303.067} C_VEL
LIN {X 0,Y 476.456,Z 487.381,A -85,B 0,C 180,E1 -7303.761,E2 -7303.761} C_VEL
LIN {X 0,Y 476.902,Z 475.731,A -85,B 0,C 180,E1 -7304.346,E2 -7304.346} C_VEL
LIN {X 0,Y 476.872,Z 467.026,A -85,B 0,C 180,E1 -7304.688,E2 -7304.688} C_VEL
LIN {X 0,Y 474.741,Z 454.169,A -85,B 0,C 180,E1 -7305.112,E2 -7305.112} C_VEL
LIN {X 0,Y 474.272,Z 451.452,A -85,B 0,C 180,E1 -7305.196,E2 -7305.196} C_VEL
LIN {X 0,Y 474.554,Z 440.975,A -85,B 0,C 180,E1 -7308.59,E2 -7308.59} C_VEL
LIN {X 0,Y 474.803,Z 431.422,A -85,B 0,C 180,E1 -7311.72,E2 -7311.72} C_VEL
LIN {X 0,Y 475.039,Z 421.738,A -85,B 0,C 180,E1 -7314.94,E2 -7314.94} C_VEL
LIN {X 0,Y 475.373,Z 413.66,A -85,B 0,C 180,E1 -7317.813,E2 -7317.813} C_VEL
LIN {X 0,Y 475.78,Z 404.535,A -85,B 0,C 180,E1 -7321.133,E2 -7321.133} C_VEL
LIN {X 0,Y 476.225,Z 396.24,A -85,B 0,C 180,E1 -7324.266,E2 -7324.266} C_VEL
LIN {X 0,Y 476.328,Z 391.417,A -85,B 0,C 180,E1 -7326.171,E2 -7326.171} C_VEL
LIN {X 0,Y 475.482,Z 386.123,A -85,B 0,C 180,E1 -7328.428,E2 -7328.428} C_VEL
LIN {X 0,Y 474.629,Z 381.366,A -85,B 0,C 180,E1 -7330.593,E2 -7330.593} C_VEL
LIN {X 0,Y 474.601,Z 381.37,A -85,B 0,C 180,E1 -7333.481,E2 -7333.481} C_VEL
LIN {X 0,Y 474.601,Z 381.37,A -85,B 0,C 180,E1 -7336.52,E2 -7336.52} C_VEL
LIN {X 0,Y 474.623,Z 381.366,A -85,B 0,C 180,E1 -7339.343,E2 -7339.343} C_VEL
LIN {X 0,Y 474.595,Z 381.37,A -85,B 0,C 180,E1 -7342.616,E2 -7342.616} C_VEL
LIN {X 0,Y 474.625,Z 381.364,A -85,B 0,C 180,E1 -7345.758,E2 -7345.758} C_VEL
LIN {X 0,Y 474.604,Z 381.369,A -85,B 0,C 180,E1 -7348.783,E2 -7348.783} C_VEL
LIN {X 0,Y 474.651,Z 381.36,A -85,B 0,C 180,E1 -7351.718,E2 -7351.718} C_VEL
LIN {X 0,Y 474.675,Z 381.36,A -85,B 0,C 180,E1 -7354.578,E2 -7354.578} C_VEL
LIN {X 0,Y 474.605,Z 381.367,A -85,B 0,C 180,E1 -7357.355,E2 -7357.355} C_VEL
LIN {X 0,Y 474.66,Z 381.361,A -85,B 0,C 180,E1 -7360.09,E2 -7360.09} C_VEL
LIN {X 0,Y 474.655,Z 381.362,A -85,B 0,C 180,E1 -7362.775,E2 -7362.775} C_VEL
LIN {X 0,Y 474.653,Z 381.361,A -85,B 0,C 180,E1 -7365.421,E2 -7365.421} C_VEL
LIN {X 0,Y 474.709,Z 381.356,A -85,B 0,C 180,E1 -7368.038,E2 -7368.038} C_VEL
LIN {X 0,Y 474.733,Z 381.35,A -85,B 0,C 180,E1 -7371.486,E2 -7371.486} C_VEL
LIN {X 0,Y 474.776,Z 381.348,A -85,B 0,C 180,E1 -7374.052,E2 -7374.052} C_VEL
LIN {X 0,Y 474.897,Z 381.331,A -85,B 0,C 180,E1 -7377.455,E2 -7377.455} C_VEL
LIN {X 0,Y 474.915,Z 381.331,A -85,B 0,C 180,E1 -7380,E2 -7380} C_VEL
LIN {X 0,Y 474.897,Z 381.331,A -85,B 0,C 180,E1 -7382.545,E2 -7382.545} C_VEL
LIN {X 0,Y 474.775,Z 381.348,A -85,B 0,C 180,E1 -7385.948,E2 -7385.948} C_VEL
LIN {X 0,Y 474.733,Z 381.351,A -85,B 0,C 180,E1 -7388.513,E2 -7388.513} C_VEL
LIN {X 0,Y 474.709,Z 381.356,A -85,B 0,C 180,E1 -7391.962,E2 -7391.962} C_VEL
LIN {X 0,Y 474.705,Z 381.356,A -85,B 0,C 180,E1 -7395.455,E2 -7395.455} C_VEL
LIN {X 0,Y 474.669,Z 381.36,A -85,B 0,C 180,E1 -7399.01,E2 -7399.01} C_VEL
LIN {X 0,Y 474.593,Z 381.371,A -85,B 0,C 180,E1 -7401.729,E2 -7401.729} C_VEL
LIN {X 0,Y 474.662,Z 381.359,A -85,B 0,C 180,E1 -7404.493,E2 -7404.493} C_VEL
LIN {X 0,Y 474.686,Z 381.359,A -85,B 0,C 180,E1 -7407.334,E2 -7407.334} C_VEL
LIN {X 0,Y 474.61,Z 381.366,A -85,B 0,C 180,E1 -7410.23,E2 -7410.23} C_VEL
LIN {X 0,Y 474.648,Z 381.364,A -85,B 0,C 180,E1 -7413.22,E2 -7413.22} C_VEL
LIN {X 0,Y 474.593,Z 381.368,A -85,B 0,C 180,E1 -7416.323,E2 -7416.323} C_VEL
LIN {X 0,Y 474.632,Z 381.365,A -85,B 0,C 180,E1 -7419.647,E2 -7419.647} C_VEL
LIN {X 0,Y 474.619,Z 381.367,A -85,B 0,C 180,E1 -7422.934,E2 -7422.934} C_VEL
LIN {X 0,Y 474.611,Z 381.365,A -85,B 0,C 180,E1 -7425.894,E2 -7425.894} C_VEL
LIN {X 0,Y 474.633,Z 381.366,A -85,B 0,C 180,E1 -7429.04,E2 -7429.04} C_VEL
LIN {X 0,Y 474.615,Z 381.367,A -85,B 0,C 180,E1 -7431.703,E2 -7431.703} C_VEL
LIN {X 0,Y 474.63,Z 381.365,A -85,B 0,C 180,E1 -7434.725,E2 -7434.725} C_VEL
LIN {X 0,Y 474.641,Z 381.363,A -85,B 0,C 180,E1 -7437.787,E2 -7437.787} C_VEL
LIN {X 0,Y 474.628,Z 381.366,A -85,B 0,C 180,E1 -7440.884,E2 -7440.884} C_VEL
LIN {X 0,Y 474.665,Z 381.358,A -85,B 0,C 180,E1 -7443.627,E2 -7443.627} C_VEL
LIN {X 0,Y 474.641,Z 381.365,A -85,B 0,C 180,E1 -7446.64,E2 -7446.64} C_VEL
LIN {X 0,Y 474.66,Z 381.36,A -85,B 0,C 180,E1 -7450.088,E2 -7450.088} C_VEL
LIN {X 0,Y 474.659,Z 381.36,A -85,B 0,C 180,E1 -7451.672,E2 -7451.672} C_VEL
LIN {X 0,Y 473.995,Z 381.445,A -85,B 0,C 180,E1 -7452.381,E2 -7452.381} C_VEL
LIN {X 0,Y 471.145,Z 381.8,A -85,B 0,C 180,E1 -7453.533,E2 -7453.533} C_VEL
LIN {X 0,Y 468.729,Z 382.1,A -85,B 0,C 180,E1 -7454.461,E2 -7454.461} C_VEL
LIN {X 0,Y 467.687,Z 382.229,A -85,B 0,C 180,E1 -7455.178,E2 -7455.178} C_VEL
LIN {X 0,Y 467.599,Z 382.239,A -85,B 0,C 180,E1 -7455.421,E2 -7455.421} C_VEL
LIN {X 0,Y 467.617,Z 382.238,A -85,B 0,C 180,E1 -7457.852,E2 -7457.852} C_VEL
LIN {X 0,Y 467.195,Z 382.378,A -85,B 0,C 180,E1 -7461.347,E2 -7461.347} C_VEL
LIN {X 0,Y 467.12,Z 385.08,A -85,B 0,C 180,E1 -7463.953,E2 -7463.953} C_VEL
LIN {X 0,Y 467.241,Z 386.88,A -85,B 0,C 180,E1 -7465.685,E2 -7465.685} C_VEL
LIN {X 0,Y 466.935,Z 391.459,A -85,B 0,C 180,E1 -7469.998,E2 -7469.998} C_VEL
LIN {X 0,Y 467.002,Z 395.19,A -85,B 0,C 180,E1 -7473.449,E2 -7473.449} C_VEL
LIN {X 0,Y 466.917,Z 398.917,A -85,B 0,C 180,E1 -7476.914,E2 -7476.914} C_VEL
LIN {X 0,Y 466.864,Z 399.778,A -85,B 0,C 180,E1 -7477.703,E2 -7477.703} C_VEL
LIN {X 0,Y 470.185,Z 414.32,A -85,B 0,C 180,E1 -7478.27,E2 -7478.27} C_VEL
LIN {X 0,Y 470.071,Z 425.333,A -85,B 0,C 180,E1 -7478.763,E2 -7478.763} C_VEL
LIN {X 0,Y 469.588,Z 437.405,A -85,B 0,C 180,E1 -7479.474,E2 -7479.474} C_VEL
LIN {X 0,Y 469.193,Z 447.628,A -85,B 0,C 180,E1 -7480.244,E2 -7480.244} C_VEL
LIN {X 0,Y 468.656,Z 458.293,A -85,B 0,C 180,E1 -7481.24,E2 -7481.24} C_VEL
LIN {X 0,Y 468.208,Z 467.38,A -85,B 0,C 180,E1 -7482.287,E2 -7482.287} C_VEL
LIN {X 0,Y 467.77,Z 475.693,A -85,B 0,C 180,E1 -7483.465,E2 -7483.465} C_VEL
LIN {X 0,Y 467.431,Z 483.336,A -85,B 0,C 180,E1 -7484.807,E2 -7484.807} C_VEL
LIN {X 0,Y 467.162,Z 489.289,A -85,B 0,C 180,E1 -7486.113,E2 -7486.113} C_VEL
LIN {X 0,Y 466.952,Z 494.313,A -85,B 0,C 180,E1 -7487.517,E2 -7487.517} C_VEL
LIN {X 0,Y 466.838,Z 496.992,A -85,B 0,C 180,E1 -7488.48,E2 -7488.48} C_VEL
LIN {X 0,Y 466.743,Z 498.935,A -85,B 0,C 180,E1 -7489.343,E2 -7489.343} C_VEL
LIN {X 0,Y 466.654,Z 501.477,A -85,B 0,C 180,E1 -7490.974,E2 -7490.974} C_VEL
LIN {X 0,Y 466.615,Z 502.368,A -85,B 0,C 180,E1 -7492.117,E2 -7492.117} C_VEL
LIN {X 0,Y 466.629,Z 502.592,A -85,B 0,C 180,E1 -7493.258,E2 -7493.258} C_VEL
LIN {X 0,Y 466.64,Z 501.678,A -85,B 0,C 180,E1 -7494.94,E2 -7494.94} C_VEL
LIN {X 0,Y 466.682,Z 500.504,A -85,B 0,C 180,E1 -7495.893,E2 -7495.893} C_VEL
LIN {X 0,Y 466.842,Z 497.7,A -85,B 0,C 180,E1 -7497.351,E2 -7497.351} C_VEL
LIN {X 0,Y 466.984,Z 493.726,A -85,B 0,C 180,E1 -7498.787,E2 -7498.787} C_VEL
LIN {X 0,Y 467.229,Z 488.275,A -85,B 0,C 180,E1 -7500.256,E2 -7500.256} C_VEL
LIN {X 0,Y 467.528,Z 482.223,A -85,B 0,C 180,E1 -7501.533,E2 -7501.533} C_VEL
LIN {X 0,Y 467.867,Z 475.205,A -85,B 0,C 180,E1 -7502.733,E2 -7502.733} C_VEL
LIN {X 0,Y 468.315,Z 466.409,A -85,B 0,C 180,E1 -7503.949,E2 -7503.949} C_VEL
LIN {X 0,Y 468.801,Z 455.936,A -85,B 0,C 180,E1 -7505.118,E2 -7505.118} C_VEL
LIN {X 0,Y 469.308,Z 445.647,A -85,B 0,C 180,E1 -7506.034,E2 -7506.034} C_VEL
LIN {X 0,Y 469.805,Z 433.524,A -85,B 0,C 180,E1 -7506.884,E2 -7506.884} C_VEL
LIN {X 0,Y 470.2,Z 421.745,A -85,B 0,C 180,E1 -7507.518,E2 -7507.518} C_VEL
LIN {X 0,Y 470.351,Z 415.735,A -85,B 0,C 180,E1 -7507.776,E2 -7507.776} C_VEL
LIN {X 0,Y 467.92,Z 404.681,A -85,B 0,C 180,E1 -7508.236,E2 -7508.236} C_VEL
LIN {X 0,Y 466.833,Z 400.204,A -85,B 0,C 180,E1 -7508.404,E2 -7508.404} C_VEL
LIN {X 0,Y 466.847,Z 396.95,A -85,B 0,C 180,E1 -7511.479,E2 -7511.479} C_VEL
LIN {X 0,Y 466.952,Z 394.472,A -85,B 0,C 180,E1 -7513.812,E2 -7513.812} C_VEL
LIN {X 0,Y 466.996,Z 391.946,A -85,B 0,C 180,E1 -7516.247,E2 -7516.247} C_VEL
LIN {X 0,Y 467.025,Z 388.386,A -85,B 0,C 180,E1 -7519.678,E2 -7519.678} C_VEL
LIN {X 0,Y 467.133,Z 384.972,A -85,B 0,C 180,E1 -7523.001,E2 -7523.001} C_VEL
LIN {X 0,Y 467.229,Z 382.29,A -85,B 0,C 180,E1 -7525.818,E2 -7525.818} C_VEL
LIN {X 0,Y 467.521,Z 382.251,A -85,B 0,C 180,E1 -7528.96,E2 -7528.96} C_VEL
LIN {X 0,Y 467.61,Z 382.24,A -85,B 0,C 180,E1 -7532.23,E2 -7532.23} C_VEL
LIN {X 0,Y 467.598,Z 382.244,A -85,B 0,C 180,E1 -7535.112,E2 -7535.112} C_VEL
LIN {X 0,Y 467.559,Z 382.247,A -85,B 0,C 180,E1 -7537.927,E2 -7537.927} C_VEL
LIN {X 0,Y 467.605,Z 382.24,A -85,B 0,C 180,E1 -7540.691,E2 -7540.691} C_VEL
LIN {X 0,Y 467.629,Z 382.235,A -85,B 0,C 180,E1 -7544.114,E2 -7544.114} C_VEL
LIN {X 0,Y 467.662,Z 382.231,A -85,B 0,C 180,E1 -7547.855,E2 -7547.855} C_VEL
LIN {X 0,Y 467.663,Z 382.234,A -85,B 0,C 180,E1 -7551.357,E2 -7551.357} C_VEL
LIN {X 0,Y 467.735,Z 382.224,A -85,B 0,C 180,E1 -7553.963,E2 -7553.963} C_VEL
LIN {X 0,Y 467.843,Z 382.208,A -85,B 0,C 180,E1 -7557.417,E2 -7557.417} C_VEL
LIN {X 0,Y 467.861,Z 382.206,A -85,B 0,C 180,E1 -7560,E2 -7560} C_VEL
LIN {X 0,Y 467.849,Z 382.208,A -85,B 0,C 180,E1 -7562.583,E2 -7562.583} C_VEL
LIN {X 0,Y 467.724,Z 382.226,A -85,B 0,C 180,E1 -7566.038,E2 -7566.038} C_VEL
LIN {X 0,Y 467.662,Z 382.233,A -85,B 0,C 180,E1 -7568.643,E2 -7568.643} C_VEL
LIN {X 0,Y 467.662,Z 382.231,A -85,B 0,C 180,E1 -7572.145,E2 -7572.145} C_VEL
LIN {X 0,Y 467.629,Z 382.237,A -85,B 0,C 180,E1 -7575.886,E2 -7575.886} C_VEL
LIN {X 0,Y 467.605,Z 382.239,A -85,B 0,C 180,E1 -7579.309,E2 -7579.309} C_VEL
LIN {X 0,Y 467.56,Z 382.246,A -85,B 0,C 180,E1 -7582.073,E2 -7582.073} C_VEL
LIN {X 0,Y 467.599,Z 382.243,A -85,B 0,C 180,E1 -7584.888,E2 -7584.888} C_VEL
LIN {X 0,Y 467.609,Z 382.243,A -85,B 0,C 180,E1 -7587.77,E2 -7587.77} C_VEL
LIN {X 0,Y 467.552,Z 382.247,A -85,B 0,C 180,E1 -7591.047,E2 -7591.047} C_VEL
LIN {X 0,Y 467.574,Z 382.244,A -85,B 0,C 180,E1 -7594.244,E2 -7594.244} C_VEL
LIN {X 0,Y 467.537,Z 382.25,A -85,B 0,C 180,E1 -7597.189,E2 -7597.189} C_VEL
LIN {X 0,Y 467.583,Z 382.245,A -85,B 0,C 180,E1 -7600.264,E2 -7600.264} C_VEL
LIN {X 0,Y 467.606,Z 382.245,A -85,B 0,C 180,E1 -7602.573,E2 -7602.573} C_VEL
LIN {X 0,Y 467.562,Z 382.25,A -85,B 0,C 180,E1 -7606.178,E2 -7606.178} C_VEL
LIN {X 0,Y 467.595,Z 382.288,A -85,B 0,C 180,E1 -7609.174,E2 -7609.174} C_VEL
LIN {X 0,Y 468.964,Z 389.708,A -85,B 0,C 180,E1 -7612.587,E2 -7612.587} C_VEL
LIN {X 0,Y 469.342,Z 393.593,A -85,B 0,C 180,E1 -7614.271,E2 -7614.271} C_VEL
LIN {X 0,Y 469.012,Z 400.65,A -85,B 0,C 180,E1 -7617.05,E2 -7617.05} C_VEL
LIN {X 0,Y 468.581,Z 408.047,A -85,B 0,C 180,E1 -7619.84,E2 -7619.84} C_VEL
LIN {X 0,Y 468.241,Z 416.084,A -85,B 0,C 180,E1 -7622.774,E2 -7622.774} C_VEL
LIN {X 0,Y 467.954,Z 424.035,A -85,B 0,C 180,E1 -7625.608,E2 -7625.608} C_VEL
LIN {X 0,Y 467.656,Z 433.741,A -85,B 0,C 180,E1 -7628.861,E2 -7628.861} C_VEL
LIN {X 0,Y 467.392,Z 443.401,A -85,B 0,C 180,E1 -7632.048,E2 -7632.048} C_VEL
LIN {X 0,Y 467.23,Z 451.115,A -85,B 0,C 180,E1 -7634.573,E2 -7634.573} C_VEL
LIN {X 0,Y 469.742,Z 466.37,A -85,B 0,C 180,E1 -7635.073,E2 -7635.073} C_VEL
LIN {X 0,Y 470.193,Z 470.227,A -85,B 0,C 180,E1 -7635.226,E2 -7635.226} C_VEL
LIN {X 0,Y 469.723,Z 483.264,A -85,B 0,C 180,E1 -7635.82,E2 -7635.82} C_VEL
LIN {X 0,Y 469.254,Z 494.492,A -85,B 0,C 180,E1 -7636.502,E2 -7636.502} C_VEL
LIN {X 0,Y 468.849,Z 505.127,A -85,B 0,C 180,E1 -7637.318,E2 -7637.318} C_VEL
LIN {X 0,Y 468.395,Z 515.613,A -85,B 0,C 180,E1 -7638.315,E2 -7638.315} C_VEL
LIN {X 0,Y 467.877,Z 524.799,A -85,B 0,C 180,E1 -7639.399,E2 -7639.399} C_VEL
LIN {X 0,Y 467.445,Z 533.699,A -85,B 0,C 180,E1 -7640.701,E2 -7640.701} C_VEL
LIN {X 0,Y 467.091,Z 540.857,A -85,B 0,C 180,E1 -7642.002,E2 -7642.002} C_VEL
LIN {X 0,Y 466.906,Z 547.077,A -85,B 0,C 180,E1 -7643.44,E2 -7643.44} C_VEL
LIN {X 0,Y 466.783,Z 551.682,A -85,B 0,C 180,E1 -7644.819,E2 -7644.819} C_VEL
LIN {X 0,Y 466.662,Z 553.962,A -85,B 0,C 180,E1 -7645.683,E2 -7645.683} C_VEL
